# B&R Automation Studio project TD52 (part 18)

```c
/* Source: zlanhe.f */
#define zlanhe FORTRAN_WRAPPER(zlanhe)
extern double zlanhe(
    char   *norm,
    char   *uplo,
    ptrdiff_t *n,
    double *a,
    ptrdiff_t *lda,
    double *work
);

/* Source: zlanhf.f */
#define zlanhf FORTRAN_WRAPPER(zlanhf)
extern double zlanhf(
    char   *norm,
    char   *transr,
    char   *uplo,
    ptrdiff_t *n,
    double *a,
    double *work
);

/* Source: zlanhp.f */
#define zlanhp FORTRAN_WRAPPER(zlanhp)
extern double zlanhp(
    char   *norm,
    char   *uplo,
    ptrdiff_t *n,
    double *ap,
    double *work
);

/* Source: zlanhs.f */
#define zlanhs FORTRAN_WRAPPER(zlanhs)
extern double zlanhs(
    char   *norm,
    ptrdiff_t *n,
    double *a,
    ptrdiff_t *lda,
    double *work
);

/* Source: zlanht.f */
#define zlanht FORTRAN_WRAPPER(zlanht)
extern double zlanht(
    char   *norm,
    ptrdiff_t *n,
    double *d,
    double *e
);

/* Source: zlansb.f */
#define zlansb FORTRAN_WRAPPER(zlansb)
extern double zlansb(
    char   *norm,
    char   *uplo,
    ptrdiff_t *n,
    ptrdiff_t *k,
    double *ab,
    ptrdiff_t *ldab,
    double *work
);

/* Source: zlansp.f */
#define zlansp FORTRAN_WRAPPER(zlansp)
extern double zlansp(
    char   *norm,
    char   *uplo,
    ptrdiff_t *n,
    double *ap,
    double *work
);

/* Source: zlansy.f */
#define zlansy FORTRAN_WRAPPER(zlansy)
extern double zlansy(
    char   *norm,
    char   *uplo,
    ptrdiff_t *n,
    double *a,
    ptrdiff_t *lda,
    double *work
);

/* Source: zlantb.f */
#define zlantb FORTRAN_WRAPPER(zlantb)
extern double zlantb(
    char   *norm,
    char   *uplo,
    char   *diag,
    ptrdiff_t *n,
    ptrdiff_t *k,
    double *ab,
    ptrdiff_t *ldab,
    double *work
);

/* Source: zlantp.f */
#define zlantp FORTRAN_WRAPPER(zlantp)
extern double zlantp(
    char   *norm,
    char   *uplo,
    char   *diag,
    ptrdiff_t *n,
    double *ap,
    double *work
);

/* Source: zlantr.f */
#define zlantr FORTRAN_WRAPPER(zlantr)
extern double zlantr(
    char   *norm,
    char   *uplo,
    char   *diag,
    ptrdiff_t *m,
    ptrdiff_t *n,
    double *a,
    ptrdiff_t *lda,
    double *work
);

/* Source: zlapll.f */
#define zlapll FORTRAN_WRAPPER(zlapll)
extern void zlapll(
    ptrdiff_t *n,
    double *x,
    ptrdiff_t *incx,
    double *y,
    ptrdiff_t *incy,
    double *ssmin
);

/* Source: zlapmt.f */
#define zlapmt FORTRAN_WRAPPER(zlapmt)
extern void zlapmt(
    ptrdiff_t *forwrd,
    ptrdiff_t *m,
    ptrdiff_t *n,
    double *x,
    ptrdiff_t *ldx,
    ptrdiff_t *k
);

/* Source: zlaqgb.f */
#define zlaqgb FORTRAN_WRAPPER(zlaqgb)
extern void zlaqgb(
    ptrdiff_t *m,
    ptrdiff_t *n,
    ptrdiff_t *kl,
    ptrdiff_t *ku,
    double *ab,
    ptrdiff_t *ldab,
    double *r,
    double *c,
    double *rowcnd,
    double *colcnd,
    double *amax,
    char   *equed
);

/* Source: zlaqge.f */
#define zlaqge FORTRAN_WRAPPER(zlaqge)
extern void zlaqge(
    ptrdiff_t *m,
    ptrdiff_t *n,
    double *a,
    ptrdiff_t *lda,
    double *r,
    double *c,
    double *rowcnd,
    double *colcnd,
    double *amax,
    char   *equed
);

/* Source: zlaqhb.f */
#define zlaqhb FORTRAN_WRAPPER(zlaqhb)
extern void zlaqhb(
    char   *uplo,
    ptrdiff_t *n,
    ptrdiff_t *kd,
    double *ab,
    ptrdiff_t *ldab,
    double *s,
    double *scond,
    double *amax,
    char   *equed
);

/* Source: zlaqhe.f */
#define zlaqhe FORTRAN_WRAPPER(zlaqhe)
extern void zlaqhe(
    char   *uplo,
    ptrdiff_t *n,
    double *a,
    ptrdiff_t *lda,
    double *s,
    double *scond,
    double *amax,
    char   *equed
);

/* Source: zlaqhp.f */
#define zlaqhp FORTRAN_WRAPPER(zlaqhp)
extern void zlaqhp(
    char   *uplo,
    ptrdiff_t *n,
    double *ap,
    double *s,
    double *scond,
    double *amax,
    char   *equed
);

/* Source: zlaqp2.f */
#define zlaqp2 FORTRAN_WRAPPER(zlaqp2)
extern void zlaqp2(
    ptrdiff_t *m,
    ptrdiff_t *n,
    ptrdiff_t *offset,
    double *a,
    ptrdiff_t *lda,
    ptrdiff_t *jpvt,
    double *tau,
    double *vn1,
    double *vn2,
    double *work
);

/* Source: zlaqps.f */
#define zlaqps FORTRAN_WRAPPER(zlaqps)
extern void zlaqps(
    ptrdiff_t *m,
    ptrdiff_t *n,
    ptrdiff_t *offset,
    ptrdiff_t *nb,
    ptrdiff_t *kb,
    double *a,
    ptrdiff_t *lda,
    ptrdiff_t *jpvt,
    double *tau,
    double *vn1,
    double *vn2,
    double *auxv,
    double *f,
    ptrdiff_t *ldf
);

/* Source: zlaqr0.f */
#define zlaqr0 FORTRAN_WRAPPER(zlaqr0)
extern void zlaqr0(
    ptrdiff_t *wantt,
    ptrdiff_t *wantz,
    ptrdiff_t *n,
    ptrdiff_t *ilo,
    ptrdiff_t *ihi,
    double *h,
    ptrdiff_t *ldh,
    double *w,
    ptrdiff_t *iloz,
    ptrdiff_t *ihiz,
    double *z,
    ptrdiff_t *ldz,
    double *work,
    ptrdiff_t *lwork,
    ptrdiff_t *info
);

/* Source: zlaqr1.f */
#define zlaqr1 FORTRAN_WRAPPER(zlaqr1)
extern void zlaqr1(
    ptrdiff_t *n,
    double *h,
    ptrdiff_t *ldh,
    double *s1,
    double *s2,
    double *v
);

/* Source: zlaqr2.f */
#define zlaqr2 FORTRAN_WRAPPER(zlaqr2)
extern void zlaqr2(
    ptrdiff_t *wantt,
    ptrdiff_t *wantz,
    ptrdiff_t *n,
    ptrdiff_t *ktop,
    ptrdiff_t *kbot,
    ptrdiff_t *nw,
    double *h,
    ptrdiff_t *ldh,
    ptrdiff_t *iloz,
    ptrdiff_t *ihiz,
    double *z,
    ptrdiff_t *ldz,
    ptrdiff_t *ns,
    ptrdiff_t *nd,
    double *sh,
    double *v,
    ptrdiff_t *ldv,
    ptrdiff_t *nh,
    double *t,
    ptrdiff_t *ldt,
    ptrdiff_t *nv,
    double *wv,
    ptrdiff_t *ldwv,
    double *work,
    ptrdiff_t *lwork
);

/* Source: zlaqr3.f */
#define zlaqr3 FORTRAN_WRAPPER(zlaqr3)
extern void zlaqr3(
    ptrdiff_t *wantt,
    ptrdiff_t *wantz,
    ptrdiff_t *n,
    ptrdiff_t *ktop,
    ptrdiff_t *kbot,
    ptrdiff_t *nw,
    double *h,
    ptrdiff_t *ldh,
    ptrdiff_t *iloz,
    ptrdiff_t *ihiz,
    double *z,
    ptrdiff_t *ldz,
    ptrdiff_t *ns,
    ptrdiff_t *nd,
    double *sh,
    double *v,
    ptrdiff_t *ldv,
    ptrdiff_t *nh,
    double *t,
    ptrdiff_t *ldt,
    ptrdiff_t *nv,
    double *wv,
    ptrdiff_t *ldwv,
    double *work,
    ptrdiff_t *lwork
);

/* Source: zlaqr4.f */
#define zlaqr4 FORTRAN_WRAPPER(zlaqr4)
extern void zlaqr4(
    ptrdiff_t *wantt,
    ptrdiff_t *wantz,
    ptrdiff_t *n,
    ptrdiff_t *ilo,
    ptrdiff_t *ihi,
    double *h,
    ptrdiff_t *ldh,
    double *w,
    ptrdiff_t *iloz,
    ptrdiff_t *ihiz,
    double *z,
    ptrdiff_t *ldz,
    double *work,
    ptrdiff_t *lwork,
    ptrdiff_t *info
);

/* Source: zlaqr5.f */
#define zlaqr5 FORTRAN_WRAPPER(zlaqr5)
extern void zlaqr5(
    ptrdiff_t *wantt,
    ptrdiff_t *wantz,
    ptrdiff_t *kacc22,
    ptrdiff_t *n,
    ptrdiff_t *ktop,
    ptrdiff_t *kbot,
    ptrdiff_t *nshfts,
    double *s,
    double *h,
    ptrdiff_t *ldh,
    ptrdiff_t *iloz,
    ptrdiff_t *ihiz,
    double *z,
    ptrdiff_t *ldz,
    double *v,
    ptrdiff_t *ldv,
    double *u,
    ptrdiff_t *ldu,
    ptrdiff_t *nv,
    double *wv,
    ptrdiff_t *ldwv,
    ptrdiff_t *nh,
    double *wh,
    ptrdiff_t *ldwh
);

/* Source: zlaqsb.f */
#define zlaqsb FORTRAN_WRAPPER(zlaqsb)
extern void zlaqsb(
    char   *uplo,
    ptrdiff_t *n,
    ptrdiff_t *kd,
    double *ab,
    ptrdiff_t *ldab,
    double *s,
    double *scond,
    double *amax,
    char   *equed
);

/* Source: zlaqsp.f */
#define zlaqsp FORTRAN_WRAPPER(zlaqsp)
extern void zlaqsp(
    char   *uplo,
    ptrdiff_t *n,
    double *ap,
    double *s,
    double *scond,
    double *amax,
    char   *equed
);

/* Source: zlaqsy.f */
#define zlaqsy FORTRAN_WRAPPER(zlaqsy)
extern void zlaqsy(
    char   *uplo,
    ptrdiff_t *n,
    double *a,
    ptrdiff_t *lda,
    double *s,
    double *scond,
    double *amax,
    char   *equed
);

/* Source: zlar1v.f */
#define zlar1v FORTRAN_WRAPPER(zlar1v)
extern void zlar1v(
    ptrdiff_t *n,
    ptrdiff_t *b1,
    ptrdiff_t *bn,
    double *lambda,
    double *d,
    double *l,
    double *ld,
    double *lld,
    double *pivmin,
    double *gaptol,
    double *z,
    ptrdiff_t *wantnc,
    ptrdiff_t *negcnt,
    double *ztz,
    double *mingma,
    ptrdiff_t *r,
    ptrdiff_t *isuppz,
    double *nrminv,
    double *resid,
    double *rqcorr,
    double *work
);

/* Source: zlar2v.f */
#define zlar2v FORTRAN_WRAPPER(zlar2v)
extern void zlar2v(
    ptrdiff_t *n,
    double *x,
    double *y,
    double *z,
    ptrdiff_t *incx,
    double *c,
    double *s,
    ptrdiff_t *incc
);

/* Source: zlarcm.f */
#define zlarcm FORTRAN_WRAPPER(zlarcm)
extern void zlarcm(
    ptrdiff_t *m,
    ptrdiff_t *n,
    double *a,
    ptrdiff_t *lda,
    double *b,
    ptrdiff_t *ldb,
    double *c,
    ptrdiff_t *ldc,
    double *rwork
);

/* Source: zlarf.f */
#define zlarf FORTRAN_WRAPPER(zlarf)
extern void zlarf(
    char   *side,
    ptrdiff_t *m,
    ptrdiff_t *n,
    double *v,
    ptrdiff_t *incv,
    double *tau,
    double *c,
    ptrdiff_t *ldc,
    double *work
);

/* Source: zlarfb.f */
#define zlarfb FORTRAN_WRAPPER(zlarfb)
extern void zlarfb(
    char   *side,
    char   *trans,
    char   *direct,
    char   *storev,
    ptrdiff_t *m,
    ptrdiff_t *n,
    ptrdiff_t *k,
    double *v,
    ptrdiff_t *ldv,
    double *t,
    ptrdiff_t *ldt,
    double *c,
    ptrdiff_t *ldc,
    double *work,
    ptrdiff_t *ldwork
);

/* Source: zlarfg.f */
#define zlarfg FORTRAN_WRAPPER(zlarfg)
extern void zlarfg(
    ptrdiff_t *n,
    double *alpha,
    double *x,
    ptrdiff_t *incx,
    double *tau
);

/* Source: zlarfgp.f */
#define zlarfgp FORTRAN_WRAPPER(zlarfgp)
extern void zlarfgp(
    ptrdiff_t *n,
    double *alpha,
    double *x,
    ptrdiff_t *incx,
    double *tau
);

/* Source: zlarft.f */
#define zlarft FORTRAN_WRAPPER(zlarft)
extern void zlarft(
    char   *direct,
    char   *storev,
    ptrdiff_t *n,
    ptrdiff_t *k,
    double *v,
    ptrdiff_t *ldv,
    double *tau,
    double *t,
    ptrdiff_t *ldt
);

/* Source: zlarfx.f */
#define zlarfx FORTRAN_WRAPPER(zlarfx)
extern void zlarfx(
    char   *side,
    ptrdiff_t *m,
    ptrdiff_t *n,
    double *v,
    double *tau,
    double *c,
    ptrdiff_t *ldc,
    double *work
);

/* Source: zlargv.f */
#define zlargv FORTRAN_WRAPPER(zlargv)
extern void zlargv(
    ptrdiff_t *n,
    double *x,
    ptrdiff_t *incx,
    double *y,
    ptrdiff_t *incy,
    double *c,
    ptrdiff_t *incc
);

/* Source: zlarnv.f */
#define zlarnv FORTRAN_WRAPPER(zlarnv)
extern void zlarnv(
    ptrdiff_t *idist,
    ptrdiff_t *iseed,
    ptrdiff_t *n,
    double *x
);

/* Source: zlarrv.f */
#define zlarrv FORTRAN_WRAPPER(zlarrv)
extern void zlarrv(
    ptrdiff_t *n,
    double *vl,
    double *vu,
    double *d,
    double *l,
    double *pivmin,
    ptrdiff_t *isplit,
    ptrdiff_t *m,
    ptrdiff_t *dol,
    ptrdiff_t *dou,
    double *minrgp,
    double *rtol1,
    double *rtol2,
    double *w,
    double *werr,
    double *wgap,
    ptrdiff_t *iblock,
    ptrdiff_t *indexw,
    double *gers,
    double *z,
    ptrdiff_t *ldz,
    ptrdiff_t *isuppz,
    double *work,
    ptrdiff_t *iwork,
    ptrdiff_t *info
);

/* Source: zlartg.f */
#define zlartg FORTRAN_WRAPPER(zlartg)
extern void zlartg(
    double *f,
    double *g,
    double *cs,
    double *sn,
    double *r
);

/* Source: zlartv.f */
#define zlartv FORTRAN_WRAPPER(zlartv)
extern void zlartv(
    ptrdiff_t *n,
    double *x,
    ptrdiff_t *incx,
    double *y,
    ptrdiff_t *incy,
    double *c,
    double *s,
    ptrdiff_t *incc
);

/* Source: zlarz.f */
#define zlarz FORTRAN_WRAPPER(zlarz)
extern void zlarz(
    char   *side,
    ptrdiff_t *m,
    ptrdiff_t *n,
    ptrdiff_t *l,
    double *v,
    ptrdiff_t *incv,
    double *tau,
    double *c,
    ptrdiff_t *ldc,
    double *work
);

/* Source: zlarzb.f */
#define zlarzb FORTRAN_WRAPPER(zlarzb)
extern void zlarzb(
    char   *side,
    char   *trans,
    char   *direct,
    char   *storev,
    ptrdiff_t *m,
    ptrdiff_t *n,
    ptrdiff_t *k,
    ptrdiff_t *l,
    double *v,
    ptrdiff_t *ldv,
    double *t,
    ptrdiff_t *ldt,
    double *c,
    ptrdiff_t *ldc,
    double *work,
    ptrdiff_t *ldwork
);

/* Source: zlarzt.f */
#define zlarzt FORTRAN_WRAPPER(zlarzt)
extern void zlarzt(
    char   *direct,
    char   *storev,
    ptrdiff_t *n,
    ptrdiff_t *k,
    double *v,
    ptrdiff_t *ldv,
    double *tau,
    double *t,
    ptrdiff_t *ldt
);

/* Source: zlascl.f */
#define zlascl FORTRAN_WRAPPER(zlascl)
extern void zlascl(
    char   *type,
    ptrdiff_t *kl,
    ptrdiff_t *ku,
    double *cfrom,
    double *cto,
    ptrdiff_t *m,
    ptrdiff_t *n,
    double *a,
    ptrdiff_t *lda,
    ptrdiff_t *info
);

/* Source: zlaset.f */
#define zlaset FORTRAN_WRAPPER(zlaset)
extern void zlaset(
    char   *uplo,
    ptrdiff_t *m,
    ptrdiff_t *n,
    double *alpha,
    double *beta,
    double *a,
    ptrdiff_t *lda
);

/* Source: zlasr.f */
#define zlasr FORTRAN_WRAPPER(zlasr)
extern void zlasr(
    char   *side,
    char   *pivot,
    char   *direct,
    ptrdiff_t *m,
    ptrdiff_t *n,
    double *c,
    double *s,
    double *a,
    ptrdiff_t *lda
);

/* Source: zlassq.f */
#define zlassq FORTRAN_WRAPPER(zlassq)
extern void zlassq(
    ptrdiff_t *n,
    double *x,
    ptrdiff_t *incx,
    double *scale,
    double *sumsq
);

/* Source: zlaswp.f */
#define zlaswp FORTRAN_WRAPPER(zlaswp)
extern void zlaswp(
    ptrdiff_t *n,
    double *a,
    ptrdiff_t *lda,
    ptrdiff_t *k1,
    ptrdiff_t *k2,
    ptrdiff_t *ipiv,
    ptrdiff_t *incx
);

/* Source: zlasyf.f */
#define zlasyf FORTRAN_WRAPPER(zlasyf)
extern void zlasyf(
    char   *uplo,
    ptrdiff_t *n,
    ptrdiff_t *nb,
    ptrdiff_t *kb,
    double *a,
    ptrdiff_t *lda,
    ptrdiff_t *ipiv,
    double *w,
    ptrdiff_t *ldw,
    ptrdiff_t *info
);

/* Source: zlat2c.f */
#define zlat2c FORTRAN_WRAPPER(zlat2c)
extern void zlat2c(
    char   *uplo,
    ptrdiff_t *n,
    double *a,
    ptrdiff_t *lda,
    float  *sa,
    ptrdiff_t *ldsa,
    ptrdiff_t *info
);

/* Source: zlatbs.f */
#define zlatbs FORTRAN_WRAPPER(zlatbs)
extern void zlatbs(
    char   *uplo,
    char   *trans,
    char   *diag,
    char   *normin,
    ptrdiff_t *n,
    ptrdiff_t *kd,
    double *ab,
    ptrdiff_t *ldab,
    double *x,
    double *scale,
    double *cnorm,
    ptrdiff_t *info
);

/* Source: zlatdf.f */
#define zlatdf FORTRAN_WRAPPER(zlatdf)
extern void zlatdf(
    ptrdiff_t *ijob,
    ptrdiff_t *n,
    double *z,
    ptrdiff_t *ldz,
    double *rhs,
    double *rdsum,
    double *rdscal,
    ptrdiff_t *ipiv,
    ptrdiff_t *jpiv
);

/* Source: zlatps.f */
#define zlatps FORTRAN_WRAPPER(zlatps)
extern void zlatps(
    char   *uplo,
    char   *trans,
    char   *diag,
    char   *normin,
    ptrdiff_t *n,
    double *ap,
    double *x,
    double *scale,
    double *cnorm,
    ptrdiff_t *info
);

/* Source: zlatrd.f */
#define zlatrd FORTRAN_WRAPPER(zlatrd)
extern void zlatrd(
    char   *uplo,
    ptrdiff_t *n,
    ptrdiff_t *nb,
    double *a,
    ptrdiff_t *lda,
    double *e,
    double *tau,
    double *w,
    ptrdiff_t *ldw
);

/* Source: zlatrs.f */
#define zlatrs FORTRAN_WRAPPER(zlatrs)
extern void zlatrs(
    char   *uplo,
    char   *trans,
    char   *diag,
    char   *normin,
    ptrdiff_t *n,
    double *a,
    ptrdiff_t *lda,
    double *x,
    double *scale,
    double *cnorm,
    ptrdiff_t *info
);

/* Source: zlatrz.f */
#define zlatrz FORTRAN_WRAPPER(zlatrz)
extern void zlatrz(
    ptrdiff_t *m,
    ptrdiff_t *n,
    ptrdiff_t *l,
    double *a,
    ptrdiff_t *lda,
    double *tau,
    double *work
);

/* Source: zlatzm.f */
#define zlatzm FORTRAN_WRAPPER(zlatzm)
extern void zlatzm(
    char   *side,
    ptrdiff_t *m,
    ptrdiff_t *n,
    double *v,
    ptrdiff_t *incv,
    double *tau,
    double *c1,
    double *c2,
    ptrdiff_t *ldc,
    double *work
);

/* Source: zlauu2.f */
#define zlauu2 FORTRAN_WRAPPER(zlauu2)
extern void zlauu2(
    char   *uplo,
    ptrdiff_t *n,
    double *a,
    ptrdiff_t *lda,
    ptrdiff_t *info
);

/* Source: zlauum.f */
#define zlauum FORTRAN_WRAPPER(zlauum)
extern void zlauum(
    char   *uplo,
    ptrdiff_t *n,
    double *a,
    ptrdiff_t *lda,
    ptrdiff_t *info
);

/* Source: zpbcon.f */
#define zpbcon FORTRAN_WRAPPER(zpbcon)
extern void zpbcon(
    char   *uplo,
    ptrdiff_t *n,
    ptrdiff_t *kd,
    double *ab,
    ptrdiff_t *ldab,
    double *anorm,
    double *rcond,
    double *work,
    double *rwork,
    ptrdiff_t *info
);

/* Source: zpbequ.f */
#define zpbequ FORTRAN_WRAPPER(zpbequ)
extern void zpbequ(
    char   *uplo,
    ptrdiff_t *n,
    ptrdiff_t *kd,
    double *ab,
    ptrdiff_t *ldab,
    double *s,
    double *scond,
    double *amax,
    ptrdiff_t *info
);

/* Source: zpbrfs.f */
#define zpbrfs FORTRAN_WRAPPER(zpbrfs)
extern void zpbrfs(
    char   *uplo,
    ptrdiff_t *n,
    ptrdiff_t *kd,
    ptrdiff_t *nrhs,
    double *ab,
    ptrdiff_t *ldab,
    double *afb,
    ptrdiff_t *ldafb,
    double *b,
    ptrdiff_t *ldb,
    double *x,
    ptrdiff_t *ldx,
    double *ferr,
    double *berr,
    double *work,
    double *rwork,
    ptrdiff_t *info
);

/* Source: zpbstf.f */
#define zpbstf FORTRAN_WRAPPER(zpbstf)
extern void zpbstf(
    char   *uplo,
    ptrdiff_t *n,
    ptrdiff_t *kd,
    double *ab,
    ptrdiff_t *ldab,
    ptrdiff_t *info
);

/* Source: zpbsv.f */
#define zpbsv FORTRAN_WRAPPER(zpbsv)
extern void zpbsv(
    char   *uplo,
    ptrdiff_t *n,
    ptrdiff_t *kd,
    ptrdiff_t *nrhs,
    double *ab,
    ptrdiff_t *ldab,
    double *b,
    ptrdiff_t *ldb,
    ptrdiff_t *info
);

/* Source: zpbsvx.f */
#define zpbsvx FORTRAN_WRAPPER(zpbsvx)
extern void zpbsvx(
    char   *fact,
    char   *uplo,
    ptrdiff_t *n,
    ptrdiff_t *kd,
    ptrdiff_t *nrhs,
    double *ab,
    ptrdiff_t *ldab,
    double *afb,
    ptrdiff_t *ldafb,
    char   *equed,
    double *s,
    double *b,
    ptrdiff_t *ldb,
    double *x,
    ptrdiff_t *ldx,
    double *rcond,
    double *ferr,
    double *berr,
    double *work,
    double *rwork,
    ptrdiff_t *info
);

/* Source: zpbtf2.f */
#define zpbtf2 FORTRAN_WRAPPER(zpbtf2)
extern void zpbtf2(
    char   *uplo,
    ptrdiff_t *n,
    ptrdiff_t *kd,
    double *ab,
    ptrdiff_t *ldab,
    ptrdiff_t *info
);

/* Source: zpbtrf.f */
#define zpbtrf FORTRAN_WRAPPER(zpbtrf)
extern void zpbtrf(
    char   *uplo,
    ptrdiff_t *n,
    ptrdiff_t *kd,
    double *ab,
    ptrdiff_t *ldab,
    ptrdiff_t *info
);

/* Source: zpbtrs.f */
#define zpbtrs FORTRAN_WRAPPER(zpbtrs)
extern void zpbtrs(
    char   *uplo,
    ptrdiff_t *n,
    ptrdiff_t *kd,
    ptrdiff_t *nrhs,
    double *ab,
    ptrdiff_t *ldab,
    double *b,
    ptrdiff_t *ldb,
    ptrdiff_t *info
);

/* Source: zpftrf.f */
#define zpftrf FORTRAN_WRAPPER(zpftrf)
extern void zpftrf(
    char   *transr,
    char   *uplo,
    ptrdiff_t *n,
    double *a,
    ptrdiff_t *info
);

/* Source: zpftri.f */
#define zpftri FORTRAN_WRAPPER(zpftri)
extern void zpftri(
    char   *transr,
    char   *uplo,
    ptrdiff_t *n,
    double *a,
    ptrdiff_t *info
);

/* Source: zpftrs.f */
#define zpftrs FORTRAN_WRAPPER(zpftrs)
extern void zpftrs(
    char   *transr,
    char   *uplo,
    ptrdiff_t *n,
    ptrdiff_t *nrhs,
    double *a,
    double *b,
    ptrdiff_t *ldb,
    ptrdiff_t *info
);

/* Source: zpocon.f */
#define zpocon FORTRAN_WRAPPER(zpocon)
extern void zpocon(
    char   *uplo,
    ptrdiff_t *n,
    double *a,
    ptrdiff_t *lda,
    double *anorm,
    double *rcond,
    double *work,
    double *rwork,
    ptrdiff_t *info
);

/* Source: zpoequ.f */
#define zpoequ FORTRAN_WRAPPER(zpoequ)
extern void zpoequ(
    ptrdiff_t *n,
    double *a,
    ptrdiff_t *lda,
    double *s,
    double *scond,
    double *amax,
    ptrdiff_t *info
);

/* Source: zpoequb.f */
#define zpoequb FORTRAN_WRAPPER(zpoequb)
extern void zpoequb(
    ptrdiff_t *n,
    double *a,
    ptrdiff_t *lda,
    double *s,
    double *scond,
    double *amax,
    ptrdiff_t *info
);

/* Source: zporfs.f */
#define zporfs FORTRAN_WRAPPER(zporfs)
extern void zporfs(
    char   *uplo,
    ptrdiff_t *n,
    ptrdiff_t *nrhs,
    double *a,
    ptrdiff_t *lda,
    double *af,
    ptrdiff_t *ldaf,
    double *b,
    ptrdiff_t *ldb,
    double *x,
    ptrdiff_t *ldx,
    double *ferr,
    double *berr,
    double *work,
    double *rwork,
    ptrdiff_t *info
);

/* Source: zposv.f */
#define zposv FORTRAN_WRAPPER(zposv)
extern void zposv(
    char   *uplo,
    ptrdiff_t *n,
    ptrdiff_t *nrhs,
    double *a,
    ptrdiff_t *lda,
    double *b,
    ptrdiff_t *ldb,
    ptrdiff_t *info
);

/* Source: zposvx.f */
#define zposvx FORTRAN_WRAPPER(zposvx)
extern void zposvx(
    char   *fact,
    char   *uplo,
    ptrdiff_t *n,
    ptrdiff_t *nrhs,
    double *a,
    ptrdiff_t *lda,
    double *af,
    ptrdiff_t *ldaf,
    char   *equed,
    double *s,
    double *b,
    ptrdiff_t *ldb,
    double *x,
    ptrdiff_t *ldx,
    double *rcond,
    double *ferr,
    double *berr,
    double *work,
    double *rwork,
    ptrdiff_t *info
);

/* Source: zpotf2.f */
#define zpotf2 FORTRAN_WRAPPER(zpotf2)
extern void zpotf2(
    char   *uplo,
    ptrdiff_t *n,
    double *a,
    ptrdiff_t *lda,
    ptrdiff_t *info
);

/* Source: zpotrf.f */
#define zpotrf FORTRAN_WRAPPER(zpotrf)
extern void zpotrf(
    char   *uplo,
    ptrdiff_t *n,
    double *a,
    ptrdiff_t *lda,
    ptrdiff_t *info
);

/* Source: zpotri.f */
#define zpotri FORTRAN_WRAPPER(zpotri)
extern void zpotri(
    char   *uplo,
    ptrdiff_t *n,
    double *a,
    ptrdiff_t *lda,
    ptrdiff_t *info
);

/* Source: zpotrs.f */
#define zpotrs FORTRAN_WRAPPER(zpotrs)
extern void zpotrs(
    char   *uplo,
    ptrdiff_t *n,
    ptrdiff_t *nrhs,
    double *a,
    ptrdiff_t *lda,
    double *b,
    ptrdiff_t *ldb,
    ptrdiff_t *info
);

/* Source: zppcon.f */
#define zppcon FORTRAN_WRAPPER(zppcon)
extern void zppcon(
    char   *uplo,
    ptrdiff_t *n,
    double *ap,
    double *anorm,
    double *rcond,
    double *work,
    double *rwork,
    ptrdiff_t *info
);

/* Source: zppequ.f */
#define zppequ FORTRAN_WRAPPER(zppequ)
extern void zppequ(
    char   *uplo,
    ptrdiff_t *n,
    double *ap,
    double *s,
    double *scond,
    double *amax,
    ptrdiff_t *info
);

/* Source: zpprfs.f */
#define zpprfs FORTRAN_WRAPPER(zpprfs)
extern void zpprfs(
    char   *uplo,
    ptrdiff_t *n,
    ptrdiff_t *nrhs,
    double *ap,
    double *afp,
    double *b,
    ptrdiff_t *ldb,
    double *x,
    ptrdiff_t *ldx,
    double *ferr,
    double *berr,
    double *work,
    double *rwork,
    ptrdiff_t *info
);

/* Source: zppsv.f */
#define zppsv FORTRAN_WRAPPER(zppsv)
extern void zppsv(
    char   *uplo,
    ptrdiff_t *n,
    ptrdiff_t *nrhs,
    double *ap,
    double *b,
    ptrdiff_t *ldb,
    ptrdiff_t *info
);

/* Source: zppsvx.f */
#define zppsvx FORTRAN_WRAPPER(zppsvx)
extern void zppsvx(
    char   *fact,
    char   *uplo,
    ptrdiff_t *n,
    ptrdiff_t *nrhs,
    double *ap,
    double *afp,
    char   *equed,
    double *s,
    double *b,
    ptrdiff_t *ldb,
    double *x,
    ptrdiff_t *ldx,
    double *rcond,
    double *ferr,
    double *berr,
    double *work,
    double *rwork,
    ptrdiff_t *info
);

/* Source: zpptrf.f */
#define zpptrf FORTRAN_WRAPPER(zpptrf)
extern void zpptrf(
    char   *uplo,
    ptrdiff_t *n,
    double *ap,
    ptrdiff_t *info
);

/* Source: zpptri.f */
#define zpptri FORTRAN_WRAPPER(zpptri)
extern void zpptri(
    char   *uplo,
    ptrdiff_t *n,
    double *ap,
    ptrdiff_t *info
);

/* Source: zpptrs.f */
#define zpptrs FORTRAN_WRAPPER(zpptrs)
extern void zpptrs(
    char   *uplo,
    ptrdiff_t *n,
    ptrdiff_t *nrhs,
    double *ap,
    double *b,
    ptrdiff_t *ldb,
    ptrdiff_t *info
);

/* Source: zpstf2.f */
#define zpstf2 FORTRAN_WRAPPER(zpstf2)
extern void zpstf2(
    char   *uplo,
    ptrdiff_t *n,
    double *a,
    ptrdiff_t *lda,
    ptrdiff_t *piv,
    ptrdiff_t *rank,
    double *tol,
    double *work,
    ptrdiff_t *info
);

/* Source: zpstrf.f */
#define zpstrf FORTRAN_WRAPPER(zpstrf)
extern void zpstrf(
    char   *uplo,
    ptrdiff_t *n,
    double *a,
    ptrdiff_t *lda,
    ptrdiff_t *piv,
    ptrdiff_t *rank,
    double *tol,
    double *work,
    ptrdiff_t *info
);

/* Source: zptcon.f */
#define zptcon FORTRAN_WRAPPER(zptcon)
extern void zptcon(
    ptrdiff_t *n,
    double *d,
    double *e,
    double *anorm,
    double *rcond,
    double *rwork,
    ptrdiff_t *info
);

/* Source: zpteqr.f */
#define zpteqr FORTRAN_WRAPPER(zpteqr)
extern void zpteqr(
    char   *compz,
    ptrdiff_t *n,
    double *d,
    double *e,
    double *z,
    ptrdiff_t *ldz,
    double *work,
    ptrdiff_t *info
);

/* Source: zptrfs.f */
#define zptrfs FORTRAN_WRAPPER(zptrfs)
extern void zptrfs(
    char   *uplo,
    ptrdiff_t *n,
    ptrdiff_t *nrhs,
    double *d,
    double *e,
    double *df,
    double *ef,
    double *b,
    ptrdiff_t *ldb,
    double *x,
    ptrdiff_t *ldx,
    double *ferr,
    double *berr,
    double *work,
    double *rwork,
    ptrdiff_t *info
);

/* Source: zptsv.f */
#define zptsv FORTRAN_WRAPPER(zptsv)
extern void zptsv(
    ptrdiff_t *n,
    ptrdiff_t *nrhs,
    double *d,
    double *e,
    double *b,
    ptrdiff_t *ldb,
    ptrdiff_t *info
);

/* Source: zptsvx.f */
#define zptsvx FORTRAN_WRAPPER(zptsvx)
extern void zptsvx(
    char   *fact,
    ptrdiff_t *n,
    ptrdiff_t *nrhs,
    double *d,
    double *e,
    double *df,
    double *ef,
    double *b,
    ptrdiff_t *ldb,
    double *x,
    ptrdiff_t *ldx,
    double *rcond,
    double *ferr,
    double *berr,
    double *work,
    double *rwork,
    ptrdiff_t *info
);

/* Source: zpttrf.f */
#define zpttrf FORTRAN_WRAPPER(zpttrf)
extern void zpttrf(
    ptrdiff_t *n,
    double *d,
    double *e,
    ptrdiff_t *info
);

/* Source: zpttrs.f */
#define zpttrs FORTRAN_WRAPPER(zpttrs)
extern void zpttrs(
    char   *uplo,
    ptrdiff_t *n,
    ptrdiff_t *nrhs,
    double *d,
    double *e,
    double *b,
    ptrdiff_t *ldb,
    ptrdiff_t *info
);

/* Source: zptts2.f */
#define zptts2 FORTRAN_WRAPPER(zptts2)
extern void zptts2(
    ptrdiff_t *iuplo,
    ptrdiff_t *n,
    ptrdiff_t *nrhs,
    double *d,
    double *e,
    double *b,
    ptrdiff_t *ldb
);

/* Source: zrot.f */
#define zrot FORTRAN_WRAPPER(zrot)
extern void zrot(
    ptrdiff_t *n,
    double *cx,
    ptrdiff_t *incx,
    double *cy,
    ptrdiff_t *incy,
    double *c,
    double *s
);

/* Source: zspcon.f */
#define zspcon FORTRAN_WRAPPER(zspcon)
extern void zspcon(
    char   *uplo,
    ptrdiff_t *n,
    double *ap,
    ptrdiff_t *ipiv,
    double *anorm,
    double *rcond,
    double *work,
    ptrdiff_t *info
);

/* Source: zspmv.f */
#define zspmv FORTRAN_WRAPPER(zspmv)
extern void zspmv(
    char   *uplo,
    ptrdiff_t *n,
    double *alpha,
    double *ap,
    double *x,
    ptrdiff_t *incx,
    double *beta,
    double *y,
    ptrdiff_t *incy
);

/* Source: zspr.f */
#define zspr FORTRAN_WRAPPER(zspr)
extern void zspr(
    char   *uplo,
    ptrdiff_t *n,
    double *alpha,
    double *x,
    ptrdiff_t *incx,
    double *ap
);

/* Source: zsprfs.f */
#define zsprfs FORTRAN_WRAPPER(zsprfs)
extern void zsprfs(
    char   *uplo,
    ptrdiff_t *n,
    ptrdiff_t *nrhs,
    double *ap,
    double *afp,
    ptrdiff_t *ipiv,
    double *b,
    ptrdiff_t *ldb,
    double *x,
    ptrdiff_t *ldx,
    double *ferr,
    double *berr,
    double *work,
    double *rwork,
    ptrdiff_t *info
);

/* Source: zspsv.f */
#define zspsv FORTRAN_WRAPPER(zspsv)
extern void zspsv(
    char   *uplo,
    ptrdiff_t *n,
    ptrdiff_t *nrhs,
    double *ap,
    ptrdiff_t *ipiv,
    double *b,
    ptrdiff_t *ldb,
    ptrdiff_t *info
);

/* Source: zspsvx.f */
#define zspsvx FORTRAN_WRAPPER(zspsvx)
extern void zspsvx(
    char   *fact,
    char   *uplo,
    ptrdiff_t *n,
    ptrdiff_t *nrhs,
    double *ap,
    double *afp,
    ptrdiff_t *ipiv,
    double *b,
    ptrdiff_t *ldb,
    double *x,
    ptrdiff_t *ldx,
    double *rcond,
    double *ferr,
    double *berr,
    double *work,
    double *rwork,
    ptrdiff_t *info
);

/* Source: zsptrf.f */
#define zsptrf FORTRAN_WRAPPER(zsptrf)
extern void zsptrf(
    char   *uplo,
    ptrdiff_t *n,
    double *ap,
    ptrdiff_t *ipiv,
    ptrdiff_t *info
);

/* Source: zsptri.f */
#define zsptri FORTRAN_WRAPPER(zsptri)
extern void zsptri(
    char   *uplo,
    ptrdiff_t *n,
    double *ap,
    ptrdiff_t *ipiv,
    double *work,
    ptrdiff_t *info
);

/* Source: zsptrs.f */
#define zsptrs FORTRAN_WRAPPER(zsptrs)
extern void zsptrs(
    char   *uplo,
    ptrdiff_t *n,
    ptrdiff_t *nrhs,
    double *ap,
    ptrdiff_t *ipiv,
    double *b,
    ptrdiff_t *ldb,
    ptrdiff_t *info
);

/* Source: zstedc.f */
#define zstedc FORTRAN_WRAPPER(zstedc)
extern void zstedc(
    char   *compz,
    ptrdiff_t *n,
    double *d,
    double *e,
    double *z,
    ptrdiff_t *ldz,
    double *work,
    ptrdiff_t *lwork,
    double *rwork,
    ptrdiff_t *lrwork,
    ptrdiff_t *iwork,
    ptrdiff_t *liwork,
    ptrdiff_t *info
);

/* Source: zstegr.f */
#define zstegr FORTRAN_WRAPPER(zstegr)
extern void zstegr(
    char   *jobz,
    char   *range,
    ptrdiff_t *n,
    double *d,
    double *e,
    double *vl,
    double *vu,
    ptrdiff_t *il,
    ptrdiff_t *iu,
    double *abstol,
    ptrdiff_t *m,
    double *w,
    double *z,
    ptrdiff_t *ldz,
    ptrdiff_t *isuppz,
    double *work,
    ptrdiff_t *lwork,
    ptrdiff_t *iwork,
    ptrdiff_t *liwork,
    ptrdiff_t *info
);

/* Source: zstein.f */
#define zstein FORTRAN_WRAPPER(zstein)
extern void zstein(
    ptrdiff_t *n,
    double *d,
    double *e,
    ptrdiff_t *m,
    double *w,
    ptrdiff_t *iblock,
    ptrdiff_t *isplit,
    double *z,
    ptrdiff_t *ldz,
    double *work,
    ptrdiff_t *iwork,
    ptrdiff_t *ifail,
    ptrdiff_t *info
);

/* Source: zstemr.f */
#define zstemr FORTRAN_WRAPPER(zstemr)
extern void zstemr(
    char   *jobz,
    char   *range,
    ptrdiff_t *n,
    double *d,
    double *e,
    double *vl,
    double *vu,
    ptrdiff_t *il,
    ptrdiff_t *iu,
    ptrdiff_t *m,
    double *w,
    double *z,
    ptrdiff_t *ldz,
    ptrdiff_t *nzc,
    ptrdiff_t *isuppz,
    ptrdiff_t *tryrac,
    double *work,
    ptrdiff_t *lwork,
    ptrdiff_t *iwork,
    ptrdiff_t *liwork,
    ptrdiff_t *info
);

/* Source: zsteqr.f */
#define zsteqr FORTRAN_WRAPPER(zsteqr)
extern void zsteqr(
    char   *compz,
    ptrdiff_t *n,
    double *d,
    double *e,
    double *z,
    ptrdiff_t *ldz,
    double *work,
    ptrdiff_t *info
);

/* Source: zsycon.f */
#define zsycon FORTRAN_WRAPPER(zsycon)
extern void zsycon(
    char   *uplo,
    ptrdiff_t *n,
    double *a,
    ptrdiff_t *lda,
    ptrdiff_t *ipiv,
    double *anorm,
    double *rcond,
    double *work,
    ptrdiff_t *info
);

/* Source: zsyequb.f */
#define zsyequb FORTRAN_WRAPPER(zsyequb)
extern void zsyequb(
    char   *uplo,
    ptrdiff_t *n,
    double *a,
    ptrdiff_t *lda,
    double *s,
    double *scond,
    double *amax,
    double *work,
    ptrdiff_t *info
);

/* Source: zsymv.f */
#define zsymv FORTRAN_WRAPPER(zsymv)
extern void zsymv(
    char   *uplo,
    ptrdiff_t *n,
    double *alpha,
    double *a,
    ptrdiff_t *lda,
    double *x,
    ptrdiff_t *incx,
    double *beta,
    double *y,
    ptrdiff_t *incy
);

/* Source: zsyr.f */
#define zsyr FORTRAN_WRAPPER(zsyr)
extern void zsyr(
    char   *uplo,
    ptrdiff_t *n,
    double *alpha,
    double *x,
    ptrdiff_t *incx,
    double *a,
    ptrdiff_t *lda
);

/* Source: zsyrfs.f */
#define zsyrfs FORTRAN_WRAPPER(zsyrfs)
extern void zsyrfs(
    char   *uplo,
    ptrdiff_t *n,
    ptrdiff_t *nrhs,
    double *a,
    ptrdiff_t *lda,
    double *af,
    ptrdiff_t *ldaf,
    ptrdiff_t *ipiv,
    double *b,
    ptrdiff_t *ldb,
    double *x,
    ptrdiff_t *ldx,
    double *ferr,
    double *berr,
    double *work,
    double *rwork,
    ptrdiff_t *info
);

/* Source: zsysv.f */
#define zsysv FORTRAN_WRAPPER(zsysv)
extern void zsysv(
    char   *uplo,
    ptrdiff_t *n,
    ptrdiff_t *nrhs,
    double *a,
    ptrdiff_t *lda,
    ptrdiff_t *ipiv,
    double *b,
    ptrdiff_t *ldb,
    double *work,
    ptrdiff_t *lwork,
    ptrdiff_t *info
);

/* Source: zsysvx.f */
#define zsysvx FORTRAN_WRAPPER(zsysvx)
extern void zsysvx(
    char   *fact,
    char   *uplo,
    ptrdiff_t *n,
    ptrdiff_t *nrhs,
    double *a,
    ptrdiff_t *lda,
    double *af,
    ptrdiff_t *ldaf,
    ptrdiff_t *ipiv,
    double *b,
    ptrdiff_t *ldb,
    double *x,
    ptrdiff_t *ldx,
    double *rcond,
    double *ferr,
    double *berr,
    double *work,
    ptrdiff_t *lwork,
    double *rwork,
    ptrdiff_t *info
);

/* Source: zsytf2.f */
#define zsytf2 FORTRAN_WRAPPER(zsytf2)
extern void zsytf2(
    char   *uplo,
    ptrdiff_t *n,
    double *a,
    ptrdiff_t *lda,
    ptrdiff_t *ipiv,
    ptrdiff_t *info
);

/* Source: zsytrf.f */
#define zsytrf FORTRAN_WRAPPER(zsytrf)
extern void zsytrf(
    char   *uplo,
    ptrdiff_t *n,
    double *a,
    ptrdiff_t *lda,
    ptrdiff_t *ipiv,
    double *work,
    ptrdiff_t *lwork,
    ptrdiff_t *info
);

/* Source: zsytri.f */
#define zsytri FORTRAN_WRAPPER(zsytri)
extern void zsytri(
    char   *uplo,
    ptrdiff_t *n,
    double *a,
    ptrdiff_t *lda,
    ptrdiff_t *ipiv,
    double *work,
    ptrdiff_t *info
);

/* Source: zsytrs.f */
#define zsytrs FORTRAN_WRAPPER(zsytrs)
extern void zsytrs(
    char   *uplo,
    ptrdiff_t *n,
    ptrdiff_t *nrhs,
    double *a,
    ptrdiff_t *lda,
    ptrdiff_t *ipiv,
    double *b,
    ptrdiff_t *ldb,
    ptrdiff_t *info
);

/* Source: ztbcon.f */
#define ztbcon FORTRAN_WRAPPER(ztbcon)
extern void ztbcon(
    char   *norm,
    char   *uplo,
    char   *diag,
    ptrdiff_t *n,
    ptrdiff_t *kd,
    double *ab,
    ptrdiff_t *ldab,
    double *rcond,
    double *work,
    double *rwork,
    ptrdiff_t *info
);

/* Source: ztbrfs.f */
#define ztbrfs FORTRAN_WRAPPER(ztbrfs)
extern void ztbrfs(
    char   *uplo,
    char   *trans,
    char   *diag,
    ptrdiff_t *n,
    ptrdiff_t *kd,
    ptrdiff_t *nrhs,
    double *ab,
    ptrdiff_t *ldab,
    double *b,
    ptrdiff_t *ldb,
    double *x,
    ptrdiff_t *ldx,
    double *ferr,
    double *berr,
    double *work,
    double *rwork,
    ptrdiff_t *info
);

/* Source: ztbtrs.f */
#define ztbtrs FORTRAN_WRAPPER(ztbtrs)
extern void ztbtrs(
    char   *uplo,
    char   *trans,
    char   *diag,
    ptrdiff_t *n,
    ptrdiff_t *kd,
    ptrdiff_t *nrhs,
    double *ab,
    ptrdiff_t *ldab,
    double *b,
    ptrdiff_t *ldb,
    ptrdiff_t *info
);

/* Source: ztfsm.f */
#define ztfsm FORTRAN_WRAPPER(ztfsm)
extern void ztfsm(
    char   *transr,
    char   *side,
    char   *uplo,
    char   *trans,
    char   *diag,
    ptrdiff_t *m,
    ptrdiff_t *n,
    double *alpha,
    double *a,
    double *b,
    ptrdiff_t *ldb
);

/* Source: ztftri.f */
#define ztftri FORTRAN_WRAPPER(ztftri)
extern void ztftri(
    char   *transr,
    char   *uplo,
    char   *diag,
    ptrdiff_t *n,
    double *a,
    ptrdiff_t *info
);

/* Source: ztfttp.f */
#define ztfttp FORTRAN_WRAPPER(ztfttp)
extern void ztfttp(
    char   *transr,
    char   *uplo,
    ptrdiff_t *n,
    double *arf,
    double *ap,
    ptrdiff_t *info
);

/* Source: ztfttr.f */
#define ztfttr FORTRAN_WRAPPER(ztfttr)
extern void ztfttr(
    char   *transr,
    char   *uplo,
    ptrdiff_t *n,
    double *arf,
    double *a,
    ptrdiff_t *lda,
    ptrdiff_t *info
);

/* Source: ztgevc.f */
#define ztgevc FORTRAN_WRAPPER(ztgevc)
extern void ztgevc(
    char   *side,
    char   *howmny,
    ptrdiff_t *select,
    ptrdiff_t *n,
    double *s,
    ptrdiff_t *lds,
    double *p,
    ptrdiff_t *ldp,
    double *vl,
    ptrdiff_t *ldvl,
    double *vr,
    ptrdiff_t *ldvr,
    ptrdiff_t *mm,
    ptrdiff_t *m,
    double *work,
    double *rwork,
    ptrdiff_t *info
);

/* Source: ztgex2.f */
#define ztgex2 FORTRAN_WRAPPER(ztgex2)
extern void ztgex2(
    ptrdiff_t *wantq,
    ptrdiff_t *wantz,
    ptrdiff_t *n,
    double *a,
    ptrdiff_t *lda,
    double *b,
    ptrdiff_t *ldb,
    double *q,
    ptrdiff_t *ldq,
    double *z,
    ptrdiff_t *ldz,
    ptrdiff_t *j1_,
    ptrdiff_t *info
);

/* Source: ztgexc.f */
#define ztgexc FORTRAN_WRAPPER(ztgexc)
extern void ztgexc(
    ptrdiff_t *wantq,
    ptrdiff_t *wantz,
    ptrdiff_t *n,
    double *a,
    ptrdiff_t *lda,
    double *b,
    ptrdiff_t *ldb,
    double *q,
    ptrdiff_t *ldq,
    double *z,
    ptrdiff_t *ldz,
    ptrdiff_t *ifst,
    ptrdiff_t *ilst,
    ptrdiff_t *info
);

/* Source: ztgsen.f */
#define ztgsen FORTRAN_WRAPPER(ztgsen)
extern void ztgsen(
    ptrdiff_t *ijob,
    ptrdiff_t *wantq,
    ptrdiff_t *wantz,
    ptrdiff_t *select,
    ptrdiff_t *n,
    double *a,
    ptrdiff_t *lda,
    double *b,
    ptrdiff_t *ldb,
    double *alpha,
    double *beta,
    double *q,
    ptrdiff_t *ldq,
    double *z,
    ptrdiff_t *ldz,
    ptrdiff_t *m,
    double *pl,
    double *pr,
    double *dif,
    double *work,
    ptrdiff_t *lwork,
    ptrdiff_t *iwork,
    ptrdiff_t *liwork,
    ptrdiff_t *info
);

/* Source: ztgsja.f */
#define ztgsja FORTRAN_WRAPPER(ztgsja)
extern void ztgsja(
    char   *jobu,
    char   *jobv,
    char   *jobq,
    ptrdiff_t *m,
    ptrdiff_t *p,
    ptrdiff_t *n,
    ptrdiff_t *k,
    ptrdiff_t *l,
    double *a,
    ptrdiff_t *lda,
    double *b,
    ptrdiff_t *ldb,
    double *tola,
    double *tolb,
    double *alpha,
    double *beta,
    double *u,
    ptrdiff_t *ldu,
    double *v,
    ptrdiff_t *ldv,
    double *q,
    ptrdiff_t *ldq,
    double *work,
    ptrdiff_t *ncycle,
    ptrdiff_t *info
);

/* Source: ztgsna.f */
#define ztgsna FORTRAN_WRAPPER(ztgsna)
extern void ztgsna(
    char   *job,
    char   *howmny,
    ptrdiff_t *select,
    ptrdiff_t *n,
    double *a,
    ptrdiff_t *lda,
    double *b,
    ptrdiff_t *ldb,
    double *vl,
    ptrdiff_t *ldvl,
    double *vr,
    ptrdiff_t *ldvr,
    double *s,
    double *dif,
    ptrdiff_t *mm,
    ptrdiff_t *m,
    double *work,
    ptrdiff_t *lwork,
    ptrdiff_t *iwork,
    ptrdiff_t *info
);

/* Source: ztgsy2.f */
#define ztgsy2 FORTRAN_WRAPPER(ztgsy2)
extern void ztgsy2(
    char   *trans,
    ptrdiff_t *ijob,
    ptrdiff_t *m,
    ptrdiff_t *n,
    double *a,
    ptrdiff_t *lda,
    double *b,
    ptrdiff_t *ldb,
    double *c,
    ptrdiff_t *ldc,
    double *d,
    ptrdiff_t *ldd,
    double *e,
    ptrdiff_t *lde,
    double *f,
    ptrdiff_t *ldf,
    double *scale,
    double *rdsum,
    double *rdscal,
    ptrdiff_t *info
);

/* Source: ztgsyl.f */
#define ztgsyl FORTRAN_WRAPPER(ztgsyl)
extern void ztgsyl(
    char   *trans,
    ptrdiff_t *ijob,
    ptrdiff_t *m,
    ptrdiff_t *n,
    double *a,
    ptrdiff_t *lda,
    double *b,
    ptrdiff_t *ldb,
    double *c,
    ptrdiff_t *ldc,
    double *d,
    ptrdiff_t *ldd,
    double *e,
    ptrdiff_t *lde,
    double *f,
    ptrdiff_t *ldf,
    double *scale,
    double *dif,
    double *work,
    ptrdiff_t *lwork,
    ptrdiff_t *iwork,
    ptrdiff_t *info
);

/* Source: ztpcon.f */
#define ztpcon FORTRAN_WRAPPER(ztpcon)
extern void ztpcon(
    char   *norm,
    char   *uplo,
    char   *diag,
    ptrdiff_t *n,
    double *ap,
    double *rcond,
    double *work,
    double *rwork,
    ptrdiff_t *info
);

/* Source: ztprfs.f */
#define ztprfs FORTRAN_WRAPPER(ztprfs)
extern void ztprfs(
    char   *uplo,
    char   *trans,
    char   *diag,
    ptrdiff_t *n,
    ptrdiff_t *nrhs,
    double *ap,
    double *b,
    ptrdiff_t *ldb,
    double *x,
    ptrdiff_t *ldx,
    double *ferr,
    double *berr,
    double *work,
    double *rwork,
    ptrdiff_t *info
);

/* Source: ztptri.f */
#define ztptri FORTRAN_WRAPPER(ztptri)
extern void ztptri(
    char   *uplo,
    char   *diag,
    ptrdiff_t *n,
    double *ap,
    ptrdiff_t *info
);

/* Source: ztptrs.f */
#define ztptrs FORTRAN_WRAPPER(ztptrs)
extern void ztptrs(
    char   *uplo,
    char   *trans,
    char   *diag,
    ptrdiff_t *n,
    ptrdiff_t *nrhs,
    double *ap,
    double *b,
    ptrdiff_t *ldb,
    ptrdiff_t *info
);

/* Source: ztpttf.f */
#define ztpttf FORTRAN_WRAPPER(ztpttf)
extern void ztpttf(
    char   *transr,
    char   *uplo,
    ptrdiff_t *n,
    double *ap,
    double *arf,
    ptrdiff_t *info
);

/* Source: ztpttr.f */
#define ztpttr FORTRAN_WRAPPER(ztpttr)
extern void ztpttr(
    char   *uplo,
    ptrdiff_t *n,
    double *ap,
    double *a,
    ptrdiff_t *lda,
    ptrdiff_t *info
);

/* Source: ztrcon.f */
#define ztrcon FORTRAN_WRAPPER(ztrcon)
extern void ztrcon(
    char   *norm,
    char   *uplo,
    char   *diag,
    ptrdiff_t *n,
    double *a,
    ptrdiff_t *lda,
    double *rcond,
    double *work,
    double *rwork,
    ptrdiff_t *info
);

/* Source: ztrevc.f */
#define ztrevc FORTRAN_WRAPPER(ztrevc)
extern void ztrevc(
    char   *side,
    char   *howmny,
    ptrdiff_t *select,
    ptrdiff_t *n,
    double *t,
    ptrdiff_t *ldt,
    double *vl,
    ptrdiff_t *ldvl,
    double *vr,
    ptrdiff_t *ldvr,
    ptrdiff_t *mm,
    ptrdiff_t *m,
    double *work,
    double *rwork,
    ptrdiff_t *info
);

/* Source: ztrexc.f */
#define ztrexc FORTRAN_WRAPPER(ztrexc)
extern void ztrexc(
    char   *compq,
    ptrdiff_t *n,
    double *t,
    ptrdiff_t *ldt,
    double *q,
    ptrdiff_t *ldq,
    ptrdiff_t *ifst,
    ptrdiff_t *ilst,
    ptrdiff_t *info
);

/* Source: ztrrfs.f */
#define ztrrfs FORTRAN_WRAPPER(ztrrfs)
extern void ztrrfs(
    char   *uplo,
    char   *trans,
    char   *diag,
    ptrdiff_t *n,
    ptrdiff_t *nrhs,
    double *a,
    ptrdiff_t *lda,
    double *b,
    ptrdiff_t *ldb,
    double *x,
    ptrdiff_t *ldx,
    double *ferr,
    double *berr,
    double *work,
    double *rwork,
    ptrdiff_t *info
);

/* Source: ztrsen.f */
#define ztrsen FORTRAN_WRAPPER(ztrsen)
extern void ztrsen(
    char   *job,
    char   *compq,
    ptrdiff_t *select,
    ptrdiff_t *n,
    double *t,
    ptrdiff_t *ldt,
    double *q,
    ptrdiff_t *ldq,
    double *w,
    ptrdiff_t *m,
    double *s,
    double *sep,
    double *work,
    ptrdiff_t *lwork,
    ptrdiff_t *info
);

/* Source: ztrsna.f */
#define ztrsna FORTRAN_WRAPPER(ztrsna)
extern void ztrsna(
    char   *job,
    char   *howmny,
    ptrdiff_t *select,
    ptrdiff_t *n,
    double *t,
    ptrdiff_t *ldt,
    double *vl,
    ptrdiff_t *ldvl,
    double *vr,
    ptrdiff_t *ldvr,
    double *s,
    double *sep,
    ptrdiff_t *mm,
    ptrdiff_t *m,
    double *work,
    ptrdiff_t *ldwork,
    double *rwork,
    ptrdiff_t *info
);

/* Source: ztrsyl.f */
#define ztrsyl FORTRAN_WRAPPER(ztrsyl)
extern void ztrsyl(
    char   *trana,
    char   *tranb,
    ptrdiff_t *isgn,
    ptrdiff_t *m,
    ptrdiff_t *n,
    double *a,
    ptrdiff_t *lda,
    double *b,
    ptrdiff_t *ldb,
    double *c,
    ptrdiff_t *ldc,
    double *scale,
    ptrdiff_t *info
);

/* Source: ztrti2.f */
#define ztrti2 FORTRAN_WRAPPER(ztrti2)
extern void ztrti2(
    char   *uplo,
    char   *diag,
    ptrdiff_t *n,
    double *a,
    ptrdiff_t *lda,
    ptrdiff_t *info
);

/* Source: ztrtri.f */
#define ztrtri FORTRAN_WRAPPER(ztrtri)
extern void ztrtri(
    char   *uplo,
    char   *diag,
    ptrdiff_t *n,
    double *a,
    ptrdiff_t *lda,
    ptrdiff_t *info
);

/* Source: ztrtrs.f */
#define ztrtrs FORTRAN_WRAPPER(ztrtrs)
extern void ztrtrs(
    char   *uplo,
    char   *trans,
    char   *diag,
    ptrdiff_t *n,
    ptrdiff_t *nrhs,
    double *a,
    ptrdiff_t *lda,
    double *b,
    ptrdiff_t *ldb,
    ptrdiff_t *info
);

/* Source: ztrttf.f */
#define ztrttf FORTRAN_WRAPPER(ztrttf)
extern void ztrttf(
    char   *transr,
    char   *uplo,
    ptrdiff_t *n,
    double *a,
    ptrdiff_t *lda,
    double *arf,
    ptrdiff_t *info
);

/* Source: ztrttp.f */
#define ztrttp FORTRAN_WRAPPER(ztrttp)
extern void ztrttp(
    char   *uplo,
    ptrdiff_t *n,
    double *a,
    ptrdiff_t *lda,
    double *ap,
    ptrdiff_t *info
);

/* Source: ztzrqf.f */
#define ztzrqf FORTRAN_WRAPPER(ztzrqf)
extern void ztzrqf(
    ptrdiff_t *m,
    ptrdiff_t *n,
    double *a,
    ptrdiff_t *lda,
    double *tau,
    ptrdiff_t *info
);

/* Source: ztzrzf.f */
#define ztzrzf FORTRAN_WRAPPER(ztzrzf)
extern void ztzrzf(
    ptrdiff_t *m,
    ptrdiff_t *n,
    double *a,
    ptrdiff_t *lda,
    double *tau,
    double *work,
    ptrdiff_t *lwork,
    ptrdiff_t *info
);

/* Source: zung2l.f */
#define zung2l FORTRAN_WRAPPER(zung2l)
extern void zung2l(
    ptrdiff_t *m,
    ptrdiff_t *n,
    ptrdiff_t *k,
    double *a,
    ptrdiff_t *lda,
    double *tau,
    double *work,
    ptrdiff_t *info
);

/* Source: zung2r.f */
#define zung2r FORTRAN_WRAPPER(zung2r)
extern void zung2r(
    ptrdiff_t *m,
    ptrdiff_t *n,
    ptrdiff_t *k,
    double *a,
    ptrdiff_t *lda,
    double *tau,
    double *work,
    ptrdiff_t *info
);

/* Source: zungbr.f */
#define zungbr FORTRAN_WRAPPER(zungbr)
extern void zungbr(
    char   *vect,
    ptrdiff_t *m,
    ptrdiff_t *n,
    ptrdiff_t *k,
    double *a,
    ptrdiff_t *lda,
    double *tau,
    double *work,
    ptrdiff_t *lwork,
    ptrdiff_t *info
);

/* Source: zunghr.f */
#define zunghr FORTRAN_WRAPPER(zunghr)
extern void zunghr(
    ptrdiff_t *n,
    ptrdiff_t *ilo,
    ptrdiff_t *ihi,
    double *a,
    ptrdiff_t *lda,
    double *tau,
    double *work,
    ptrdiff_t *lwork,
    ptrdiff_t *info
);

/* Source: zungl2.f */
#define zungl2 FORTRAN_WRAPPER(zungl2)
extern void zungl2(
    ptrdiff_t *m,
    ptrdiff_t *n,
    ptrdiff_t *k,
    double *a,
    ptrdiff_t *lda,
    double *tau,
    double *work,
    ptrdiff_t *info
);

/* Source: zunglq.f */
#define zunglq FORTRAN_WRAPPER(zunglq)
extern void zunglq(
    ptrdiff_t *m,
    ptrdiff_t *n,
    ptrdiff_t *k,
    double *a,
    ptrdiff_t *lda,
    double *tau,
    double *work,
    ptrdiff_t *lwork,
    ptrdiff_t *info
);

/* Source: zungql.f */
#define zungql FORTRAN_WRAPPER(zungql)
extern void zungql(
    ptrdiff_t *m,
    ptrdiff_t *n,
    ptrdiff_t *k,
    double *a,
    ptrdiff_t *lda,
    double *tau,
    double *work,
    ptrdiff_t *lwork,
    ptrdiff_t *info
);

/* Source: zungqr.f */
#define zungqr FORTRAN_WRAPPER(zungqr)
extern void zungqr(
    ptrdiff_t *m,
    ptrdiff_t *n,
    ptrdiff_t *k,
    double *a,
    ptrdiff_t *lda,
    double *tau,
    double *work,
    ptrdiff_t *lwork,
    ptrdiff_t *info
);

/* Source: zungr2.f */
#define zungr2 FORTRAN_WRAPPER(zungr2)
extern void zungr2(
    ptrdiff_t *m,
    ptrdiff_t *n,
    ptrdiff_t *k,
    double *a,
    ptrdiff_t *lda,
    double *tau,
    double *work,
    ptrdiff_t *info
);

/* Source: zungrq.f */
#define zungrq FORTRAN_WRAPPER(zungrq)
extern void zungrq(
    ptrdiff_t *m,
    ptrdiff_t *n,
    ptrdiff_t *k,
    double *a,
    ptrdiff_t *lda,
    double *tau,
    double *work,
    ptrdiff_t *lwork,
    ptrdiff_t *info
);

/* Source: zungtr.f */
#define zungtr FORTRAN_WRAPPER(zungtr)
extern void zungtr(
    char   *uplo,
    ptrdiff_t *n,
    double *a,
    ptrdiff_t *lda,
    double *tau,
    double *work,
    ptrdiff_t *lwork,
    ptrdiff_t *info
);

/* Source: zunm2l.f */
#define zunm2l FORTRAN_WRAPPER(zunm2l)
extern void zunm2l(
    char   *side,
    char   *trans,
    ptrdiff_t *m,
    ptrdiff_t *n,
    ptrdiff_t *k,
    double *a,
    ptrdiff_t *lda,
    double *tau,
    double *c,
    ptrdiff_t *ldc,
    double *work,
    ptrdiff_t *info
);

/* Source: zunm2r.f */
#define zunm2r FORTRAN_WRAPPER(zunm2r)
extern void zunm2r(
    char   *side,
    char   *trans,
    ptrdiff_t *m,
    ptrdiff_t *n,
    ptrdiff_t *k,
    double *a,
    ptrdiff_t *lda,
    double *tau,
    double *c,
    ptrdiff_t *ldc,
    double *work,
    ptrdiff_t *info
);

/* Source: zunmbr.f */
#define zunmbr FORTRAN_WRAPPER(zunmbr)
extern void zunmbr(
    char   *vect,
    char   *side,
    char   *trans,
    ptrdiff_t *m,
    ptrdiff_t *n,
    ptrdiff_t *k,
    double *a,
    ptrdiff_t *lda,
    double *tau,
    double *c,
    ptrdiff_t *ldc,
    double *work,
    ptrdiff_t *lwork,
    ptrdiff_t *info
);

/* Source: zunmhr.f */
#define zunmhr FORTRAN_WRAPPER(zunmhr)
extern void zunmhr(
    char   *side,
    char   *trans,
    ptrdiff_t *m,
    ptrdiff_t *n,
    ptrdiff_t *ilo,
    ptrdiff_t *ihi,
    double *a,
    ptrdiff_t *lda,
    double *tau,
    double *c,
    ptrdiff_t *ldc,
    double *work,
    ptrdiff_t *lwork,
    ptrdiff_t *info
);

/* Source: zunml2.f */
#define zunml2 FORTRAN_WRAPPER(zunml2)
extern void zunml2(
    char   *side,
    char   *trans,
    ptrdiff_t *m,
    ptrdiff_t *n,
    ptrdiff_t *k,
    double *a,
    ptrdiff_t *lda,
    double *tau,
    double *c,
    ptrdiff_t *ldc,
    double *work,
    ptrdiff_t *info
);

/* Source: zunmlq.f */
#define zunmlq FORTRAN_WRAPPER(zunmlq)
extern void zunmlq(
    char   *side,
    char   *trans,
    ptrdiff_t *m,
    ptrdiff_t *n,
    ptrdiff_t *k,
    double *a,
    ptrdiff_t *lda,
    double *tau,
    double *c,
    ptrdiff_t *ldc,
    double *work,
    ptrdiff_t *lwork,
    ptrdiff_t *info
);

/* Source: zunmql.f */
#define zunmql FORTRAN_WRAPPER(zunmql)
extern void zunmql(
    char   *side,
    char   *trans,
    ptrdiff_t *m,
    ptrdiff_t *n,
    ptrdiff_t *k,
    double *a,
    ptrdiff_t *lda,
    double *tau,
    double *c,
    ptrdiff_t *ldc,
    double *work,
    ptrdiff_t *lwork,
    ptrdiff_t *info
);

/* Source: zunmqr.f */
#define zunmqr FORTRAN_WRAPPER(zunmqr)
extern void zunmqr(
    char   *side,
    char   *trans,
    ptrdiff_t *m,
    ptrdiff_t *n,
    ptrdiff_t *k,
    double *a,
    ptrdiff_t *lda,
    double *tau,
    double *c,
    ptrdiff_t *ldc,
    double *work,
    ptrdiff_t *lwork,
    ptrdiff_t *info
);

/* Source: zunmr2.f */
#define zunmr2 FORTRAN_WRAPPER(zunmr2)
extern void zunmr2(
    char   *side,
    char   *trans,
    ptrdiff_t *m,
    ptrdiff_t *n,
    ptrdiff_t *k,
    double *a,
    ptrdiff_t *lda,
    double *tau,
    double *c,
    ptrdiff_t *ldc,
    double *work,
    ptrdiff_t *info
);

/* Source: zunmr3.f */
#define zunmr3 FORTRAN_WRAPPER(zunmr3)
extern void zunmr3(
    char   *side,
    char   *trans,
    ptrdiff_t *m,
    ptrdiff_t *n,
    ptrdiff_t *k,
    ptrdiff_t *l,
    double *a,
    ptrdiff_t *lda,
    double *tau,
    double *c,
    ptrdiff_t *ldc,
    double *work,
    ptrdiff_t *info
);

/* Source: zunmrq.f */
#define zunmrq FORTRAN_WRAPPER(zunmrq)
extern void zunmrq(
    char   *side,
    char   *trans,
    ptrdiff_t *m,
    ptrdiff_t *n,
    ptrdiff_t *k,
    double *a,
    ptrdiff_t *lda,
    double *tau,
    double *c,
    ptrdiff_t *ldc,
    double *work,
    ptrdiff_t *lwork,
    ptrdiff_t *info
);

/* Source: zunmrz.f */
#define zunmrz FORTRAN_WRAPPER(zunmrz)
extern void zunmrz(
    char   *side,
    char   *trans,
    ptrdiff_t *m,
    ptrdiff_t *n,
    ptrdiff_t *k,
    ptrdiff_t *l,
    double *a,
    ptrdiff_t *lda,
    double *tau,
    double *c,
    ptrdiff_t *ldc,
    double *work,
    ptrdiff_t *lwork,
    ptrdiff_t *info
);

/* Source: zunmtr.f */
#define zunmtr FORTRAN_WRAPPER(zunmtr)
extern void zunmtr(
    char   *side,
    char   *uplo,
    char   *trans,
    ptrdiff_t *m,
    ptrdiff_t *n,
    double *a,
    ptrdiff_t *lda,
    double *tau,
    double *c,
    ptrdiff_t *ldc,
    double *work,
    ptrdiff_t *lwork,
    ptrdiff_t *info
);

/* Source: zupgtr.f */
#define zupgtr FORTRAN_WRAPPER(zupgtr)
extern void zupgtr(
    char   *uplo,
    ptrdiff_t *n,
    double *ap,
    double *tau,
    double *q,
    ptrdiff_t *ldq,
    double *work,
    ptrdiff_t *info
);

/* Source: zupmtr.f */
#define zupmtr FORTRAN_WRAPPER(zupmtr)
extern void zupmtr(
    char   *side,
    char   *uplo,
    char   *trans,
    ptrdiff_t *m,
    ptrdiff_t *n,
    double *ap,
    double *tau,
    double *c,
    ptrdiff_t *ldc,
    double *work,
    ptrdiff_t *info
);

#ifdef __cplusplus
    }   /* extern "C" */
#endif

#endif /* lapack_h */
```

### mat.h
```c
/*
 * PUBLISHed header for libmat, the MAT File library.
 *
 * Copyright 1984-2010 The MathWorks, Inc.
 * All Rights Reserved.
 */

#if defined(_MSC_VER)
# pragma once
#endif
#if defined(__GNUC__) && (__GNUC__ > 3 || (__GNUC__ == 3 && __GNUC_MINOR__ > 3))
# pragma once
#endif

#ifndef mat_published_c_api_h
#define mat_published_c_api_h

#ifndef EXTERN_C
#  ifdef __cplusplus
#    define EXTERN_C extern "C"
#  else
#    define EXTERN_C extern
#  endif
#endif

#ifndef LIBMAT_API
#  define LIBMAT_API
#endif

#include <stdio.h>  /* for FILE */

#include "matrix.h" /* for mxArray */

/* incomplete typedef for MATFile */
#ifdef __cplusplus
class MATFile;
#else
typedef struct MatFile_tag MATFile;
#endif

/*
 * Open a MAT-file "filename" using mode "mode".  Return
 * a pointer to a MATFile for use with other MAT API functions.
 *
 * Current valid entries for "mode" are
 * "r"    == read only.
 * "w"    == write only (deletes any existing file with name <filename>).
 * "w4"   == as "w", but create a MATLAB 4.0 MAT-file.
 * "w7.3" == as "w", but create a MATLAB 7.3 MAT-file.
 * "u"    == update.  Read and write allowed, existing file is not deleted.
 *
 * Return NULL if an error occurs.
 */
EXTERN_C LIBMAT_API MATFile* matOpen(const char *filename, const char * mode);

/*
 * Close a MAT-file opened with matOpen.
 * The pointer-to-MATfile argument is invalid, once matClose returns.
 * Return zero for success, EOF on error.
 */
EXTERN_C LIBMAT_API int matClose(MATFile *pMF);

/*
 * Return the ANSI C FILE pointer obtained when the MAT-file was opened.
 * Warning: the FILE pointer may be NULL in the case of a MAT file format
 * that does not allow access to the raw file pointer.
 */
EXTERN_C LIBMAT_API FILE * matGetFp(MATFile *pMF);

/*
 * Write array value with the specified name to the MAT-file, deleting any
 * previously existing variable with that name in the MAT-file.
 *
 * Return zero for success, nonzero for error.
 */
EXTERN_C LIBMAT_API int matPutVariable(MATFile * pMF, const char * name, const mxArray * pA);

/*
 * Write array value with the specified name to the MAT-file pMF, deleting any
 * previously existing variable in the MAT-file with the same name.
 *
 * The variable will be written such that when the MATLAB LOAD command
 * loads the variable, it will automatically place it in the
 * global workspace and establish a link to it in the local
 * workspace (as if the command "global <varname>" had been
 * issued after the variable was loaded.)
 *
 * Return zero for success, nonzero for error.
 */
EXTERN_C LIBMAT_API int matPutVariableAsGlobal(MATFile * pMF, const char * name, const mxArray * pA);

/*
 * Read the array value for the specified variable name from a MAT-file.
 *
 * Return NULL if an error occurs.
 */
EXTERN_C LIBMAT_API mxArray * matGetVariable(MATFile * pMF, const char * name);

/*
 * Read the next array value from the current file location of the MAT-file
 * pMF.  This function should only be used in conjunction with
 * matOpen and matClose.  Passing pMF to any other API functions
 * will cause matGetNextVariable() to work incorrectly.
 *
 * Return NULL if an error occurs.
 */
EXTERN_C LIBMAT_API mxArray * matGetNextVariable(MATFile *pMF, const char **nameptr);

/*
 * Read the array header of the next array value in a MAT-file.
 * This function should only be used in conjunction with
 * matOpen and matClose.  Passing pMF to any other API functions
 * will cause matGetNextVariableInfo to work incorrectly.
 *
 * See the description of matGetVariableInfo() for the definition
 * and valid uses of an array header.
 *
 * Return NULL if an error occurs.
 */
EXTERN_C LIBMAT_API mxArray * matGetNextVariableInfo(MATFile *pMF, const char **nameptr);

/*
 * Read the array header for the variable with the specified name from
 * the MAT-file.
 *
 * An array header contains all the same information as an
 * array, except that the pr, pi, ir, and jc data structures are
 * not allocated for non-recursive data types.  That is,
 * Cells, structures, and objects contain pointers to other
 * array headers, but numeric, string, and sparse arrays do not
 * contain valid data in their pr, pi, ir, or jc fields.
 *
 * The purpose of an array header is to gain fast access to
 * information about an array without reading all the array's
 * actual data.  Thus, functions such as mxGetM, mxGetN, and mxGetClassID
 * can be used with array headers, but mxGetPr, mxGetPi, mxGetIr, mxGetJc,
 * mxSetPr, mxSetPi, mxSetIr, and mxSetJc cannot.
 *
 * An array header should NEVER be returned to MATLAB (for example via the
 * MEX API), or any other non-matrix access API function that expects a
 * full mxArray (examples include engPutVariable(), matPutVariable(), and
 * mexPutVariable()).
 *
 * Return NULL if an error occurs.
 */
EXTERN_C LIBMAT_API mxArray * matGetVariableInfo(MATFile *pMF, const char * name);

/*
 * Remove a variable with with the specified name from the MAT-file pMF.
 *
 * Return zero on success, non-zero on error.
 */
EXTERN_C LIBMAT_API int matDeleteVariable(MATFile *pMF, const char *name);

/*
 * Get a list of the names of the arrays in a MAT-file.
 * The array of strings returned by this function contains "num"
 * entries.  It is allocated with one call to mxCalloc, and so
 * can (must) be freed with one call to mxFree.
 *
 * If there are no arrays in the MAT-file, return value
 * is NULL and num is set to zero.  If an error occurs,
 * return value is NULL and num is set to a negative number.
 */
EXTERN_C LIBMAT_API char ** matGetDir(MATFile * pMF, int *num);

#endif /* mat_published_c_api_h */
```

### matrix.h
```c
/*
 * @(#)matrix.h    generated by: makeheader 5.1.5  Tue May 24 21:08:01 2011
 *
 *		built from:	../../src/include/copyright.h
 *				../../src/include/pragma_interface.h
 *				include/published_version.h
 *				include/symver.h
 *				export/include/matrix/detail/published_fwd_decls.hpp
 *				alloccbk.cpp
 *				alloclst.cpp
 *				array.cpp
 *				array2.cpp
 *				arraycbk.cpp
 *				arraycpy.cpp
 *				assignmt.cpp
 *				bytestr.cpp
 *				catenate.cpp
 *				cellindex.cpp
 *				checkdim.cpp
 *				compat32.cpp
 *				conversions.cpp
 *				end.cpp
 *				errmsg.cpp
 *				error.cpp
 *				fmxapi.cpp
 *				fmxapi_700.cpp
 *				fmxapi_730.cpp
 *				funhdl.cpp
 *				grow.cpp
 *				ieee_wrap.cpp
 *				indexcpy.cpp
 *				iocbk.cpp
 *				marshal.cpp
 *				mcat.cpp
 *				mxarray_alloc.cpp
 *				mxassert.cpp
 *				mxequal.cpp
 *				mxuint128.cpp
 *				mxutil.cpp
 *				nameindex.cpp
 *				nargchk.cpp
 *				numconv.cpp
 *				opaque.cpp
 *				permute.cpp
 *				populate.cpp
 *				protected.cpp
 *				referenc.cpp
 *				resize.cpp
 *				rndcolon.cpp
 *				rootrecord_debug.cpp
 *				scopemgr.cpp
 *				strconv.cpp
 *				subserror.cpp
 *				transpose.cpp
 *				txtcmp.cpp
 *				undoc.cpp
 *				warning.cpp
 *				zbuffer.cpp
 *				include/compat_pub.h
 */

#if defined(_MSC_VER)
# pragma once
#endif
#if defined(__GNUC__) && (__GNUC__ > 3 || (__GNUC__ == 3 && __GNUC_MINOR__ > 3))
# pragma once
#endif

#ifndef matrix_h
#define matrix_h

/*
 * Copyright 1984-2003 The MathWorks, Inc.
 * All Rights Reserved.
 */

/* Copyright 2003-2006 The MathWorks, Inc. */

/* Only define EXTERN_C if it hasn't been defined already. This allows
 * individual modules to have more control over managing their exports.
 */
#ifndef EXTERN_C

#ifdef __cplusplus
  #define EXTERN_C extern "C"
#else
  #define EXTERN_C extern
#endif

#endif

/* Version 7.4.0 */
#define MX_API_VER 0x07040000

#ifndef matrix_symver_h

/*
 * PUBLISHED APIs with changes in MATLAB 7.3
 */

#if !defined(MX_COMPAT_32) || defined(MX_INTERNAL_730)

/*
 * Include this uniformly on non-Linux platforms (no .symver)
 * Include it only internal to the matrix library on Linux
 */
#if !defined(__linux__) || defined(MX_INTERNAL_730)

#ifndef mxSetProperty
# define mxSetProperty mxSetProperty_730
#endif

#ifndef mxGetProperty
# define mxGetProperty mxGetProperty_730
#endif

#ifndef mxSetField
# define mxSetField mxSetField_730
#endif

#ifndef mxSetFieldByNumber
# define mxSetFieldByNumber mxSetFieldByNumber_730
#endif

#ifndef mxGetFieldByNumber
# define mxGetFieldByNumber mxGetFieldByNumber_730
#endif

#ifndef mxGetField
# define mxGetField mxGetField_730
#endif

#ifndef mxCreateStructMatrix
# define mxCreateStructMatrix mxCreateStructMatrix_730
#endif

#ifndef mxCreateCellMatrix
# define mxCreateCellMatrix mxCreateCellMatrix_730
#endif

#ifndef mxCreateCharMatrixFromStrings
# define mxCreateCharMatrixFromStrings mxCreateCharMatrixFromStrings_730
#endif

#ifndef mxGetString
# define mxGetString mxGetString_730
#endif

#ifndef mxGetNumberOfDimensions
# define mxGetNumberOfDimensions mxGetNumberOfDimensions_730
#endif

#ifndef mxGetDimensions
# define mxGetDimensions mxGetDimensions_730
#endif

#ifndef mxSetDimensions
# define mxSetDimensions mxSetDimensions_730
#endif

#ifndef mxSetIr
# define mxSetIr mxSetIr_730
#endif

#ifndef mxGetIr
# define mxGetIr mxGetIr_730
#endif

#ifndef mxSetJc
# define mxSetJc mxSetJc_730
#endif

#ifndef mxGetJc
# define mxGetJc mxGetJc_730
#endif

#ifndef mxCreateStructArray
# define mxCreateStructArray mxCreateStructArray_730
#endif

#ifndef mxCreateCharArray
# define mxCreateCharArray mxCreateCharArray_730
#endif

#ifndef mxCreateNumericArray
# define mxCreateNumericArray mxCreateNumericArray_730
#endif

#ifndef mxCreateCellArray
# define mxCreateCellArray mxCreateCellArray_730
#endif

#ifndef mxCreateLogicalArray
# define mxCreateLogicalArray mxCreateLogicalArray_730
#endif

#ifndef mxGetCell
# define mxGetCell mxGetCell_730
#endif

#ifndef mxSetCell
# define mxSetCell mxSetCell_730
#endif

#ifndef mxSetNzmax
# define mxSetNzmax mxSetNzmax_730
#endif

#ifndef mxSetN
# define mxSetN mxSetN_730
#endif

#ifndef mxSetM
# define mxSetM mxSetM_730
#endif

#ifndef mxGetNzmax
# define mxGetNzmax mxGetNzmax_730
#endif

#ifndef mxCreateDoubleMatrix
# define mxCreateDoubleMatrix mxCreateDoubleMatrix_730
#endif

#ifndef mxCreateNumericMatrix
# define mxCreateNumericMatrix mxCreateNumericMatrix_730
#endif

#ifndef mxCreateLogicalMatrix
# define mxCreateLogicalMatrix mxCreateLogicalMatrix_730
#endif

#ifndef mxCreateSparse
# define mxCreateSparse mxCreateSparse_730
#endif

#ifndef mxCreateSparseLogicalMatrix
# define mxCreateSparseLogicalMatrix mxCreateSparseLogicalMatrix_730
#endif

#ifndef mxGetNChars
# define mxGetNChars mxGetNChars_730
#endif

#ifndef mxCreateStringFromNChars
# define mxCreateStringFromNChars mxCreateStringFromNChars_730
#endif

#ifndef mxCalcSingleSubscript
# define mxCalcSingleSubscript mxCalcSingleSubscript_730
#endif

#ifndef mxGetDimensions_fcn
# define mxGetDimensions_fcn mxGetDimensions_730
#endif

#else

#ifndef mxGetDimensions_fcn
# define mxGetDimensions_fcn mxGetDimensions
#endif

#endif /* !__linux__ || MX_INTERNAL_730 */

#else

#ifndef mxGetDimensions_fcn
# define mxGetDimensions_fcn mxGetDimensions_700
#endif

#endif /* !MX_COMPAT_32 || MX_INTERNAL_730 */

#endif /* matrix_symver_h */

/* Copyright 2008-2010 The MathWorks, Inc. */

/*
 * NOTE: The contents of this header are ultimately PUBLISHED in
 * extern/include/matrix.h.
 */

#ifndef MATHWORKS_MATRIX_DETAIL_PUBLISHED_FWD_DECLS_HPP
#define MATHWORKS_MATRIX_DETAIL_PUBLISHED_FWD_DECLS_HPP

#include <stddef.h>
#include <tmwtypes.h>

/**
 * Forward declaration for mxArray
 */
typedef struct mxArray_tag mxArray;

/**
 * Type representing the signature for MEX functions.
 */
typedef void (*mxFunctionPtr) (int nlhs, mxArray *plhs[], int nrhs, mxArray *prhs[]);

/**
 * Maximum mxArray name length
 */
#define mxMAXNAM TMW_NAME_LENGTH_MAX

/**
 * Logical type
 */
typedef bool mxLogical;

/**
 * Typedef required for Unicode support in MATLAB
 */
typedef CHAR16_T mxChar;

/**
 * Enumeration corresponding to all the valid mxArray types.
 */
typedef enum
{
    mxUNKNOWN_CLASS = 0,
    mxCELL_CLASS,
    mxSTRUCT_CLASS,
    mxLOGICAL_CLASS,
    mxCHAR_CLASS,
    mxVOID_CLASS,
    mxDOUBLE_CLASS,
    mxSINGLE_CLASS,
    mxINT8_CLASS,
    mxUINT8_CLASS,
    mxINT16_CLASS,
    mxUINT16_CLASS,
    mxINT32_CLASS,
    mxUINT32_CLASS,
    mxINT64_CLASS,
    mxUINT64_CLASS,
    mxFUNCTION_CLASS,
    mxOPAQUE_CLASS,
    mxOBJECT_CLASS, /* keep the last real item in the list */
#if defined(_LP64) || defined(_WIN64)
    mxINDEX_CLASS = mxUINT64_CLASS,
#else
    mxINDEX_CLASS = mxUINT32_CLASS,
#endif
    /* TEMPORARY AND NASTY HACK UNTIL mxSPARSE_CLASS IS COMPLETELY ELIMINATED */
    mxSPARSE_CLASS = mxVOID_CLASS /* OBSOLETE! DO NOT USE */
}
mxClassID;

/**
 * Indicates whether floating-point mxArrays are real or complex.
 */
typedef enum
{
    mxREAL,
    mxCOMPLEX
}
mxComplexity;

#endif /* MATHWORKS_MATRIX_DETAIL_PUBLISHED_FWD_DECLS_HPP */

#include <stddef.h>	/* size_t */

/*
 * allocate memory, notifying registered listener
 */
EXTERN_C void *mxMalloc(
    size_t	n		/* number of bytes */
    );

/*
 * allocate cleared memory, notifying registered listener.
 */
EXTERN_C void *mxCalloc(
    size_t	n,	/* number of objects */
    size_t	size	/* size of objects */
    );

/*
 * free memory, notifying registered listener.
 */
EXTERN_C void mxFree(void *ptr)	/* pointer to memory to be freed */;

/*
 * reallocate memory, notifying registered listener.
 */
EXTERN_C void *mxRealloc(void *ptr, size_t size);

/*
 * Return the class (catergory) of data that the array holds.
 */
EXTERN_C mxClassID mxGetClassID(const mxArray *pa);

/*
 * Get pointer to data
 */
EXTERN_C void *mxGetData(
    const mxArray *pa		/* pointer to array */
    );

/*
 * Set pointer to data
 */
EXTERN_C void mxSetData(
    mxArray *pa,		/* pointer to array */
    void  *newdata		/* pointer to data */
    );

/*
 * Determine whether the specified array contains numeric (as opposed
 * to cell or struct) data.
 */
EXTERN_C bool mxIsNumeric(const mxArray *pa);

/*
 * Determine whether the given array is a cell array.
 */
EXTERN_C bool mxIsCell(const mxArray *pa);

/*
 * Determine whether the given array's logical flag is on.
 */
EXTERN_C bool mxIsLogical(const mxArray *pa);

/*
 * Determine whether the given array contains character data.
 */
EXTERN_C bool mxIsChar(const mxArray *pa);

/*
 * Determine whether the given array is a structure array.
 */
EXTERN_C bool mxIsStruct(const mxArray *pa);

/*
 * Determine whether the given array is an opaque array.
 */
EXTERN_C bool mxIsOpaque(const mxArray *pa);

/*
 * Returns true if specified array is a function object.
 */
EXTERN_C bool mxIsFunctionHandle(const mxArray *pa);

/*
 * This function is deprecated and is preserved only for backward compatibility.
 * DO NOT USE if possible.
 * Is array user defined MATLAB v5 object
 */
EXTERN_C bool mxIsObject(
    const mxArray *pa		/* pointer to array */
    );

/*
 * Get imaginary data pointer for numeric array
 */
EXTERN_C void *mxGetImagData(
    const mxArray *pa		/* pointer to array */
    );

/*
 * Set imaginary data pointer for numeric array
 */
EXTERN_C void mxSetImagData(
    mxArray *pa,		/* pointer to array */
    void    *newdata		/* imaginary data array pointer */
    );

/*
 * Determine whether the given array contains complex data.
 */
EXTERN_C bool mxIsComplex(const mxArray *pa);

/*
 * Determine whether the given array is a sparse (as opposed to full).
 */
EXTERN_C bool mxIsSparse(const mxArray *pa);

/*
 * Determine whether the specified array represents its data as
 * double-precision floating-point numbers.
 */
EXTERN_C bool mxIsDouble(const mxArray *pa);

/*
 * Determine whether the specified array represents its data as
 * single-precision floating-point numbers.
 */
EXTERN_C bool mxIsSingle(const mxArray *pa);

/*
 * Determine whether the specified array represents its data as
 * signed 8-bit integers.
 */
EXTERN_C bool mxIsInt8(const mxArray *pa);

/*
 * Determine whether the specified array represents its data as
 * unsigned 8-bit integers.
 */
EXTERN_C bool mxIsUint8(const mxArray *pa);

/*
 * Determine whether the specified array represents its data as
 * signed 16-bit integers.
 */
EXTERN_C bool mxIsInt16(const mxArray *pa);

/*
 * Determine whether the specified array represents its data as
 * unsigned 16-bit integers.
 */
EXTERN_C bool mxIsUint16(const mxArray *pa);

/*
 * Determine whether the specified array represents its data as
 * signed 32-bit integers.
 */
EXTERN_C bool mxIsInt32(const mxArray *pa);

/*
 * Determine whether the specified array represents its data as
 * unsigned 32-bit integers.
 */
EXTERN_C bool mxIsUint32(const mxArray *pa);

/*
 * Determine whether the specified array represents its data as
 * signed 64-bit integers.
 */
EXTERN_C bool mxIsInt64(const mxArray *pa);

/*
 * Determine whether the specified array represents its data as
 * unsigned 64-bit integers.
 */
EXTERN_C bool mxIsUint64(const mxArray *pa);

/*
 * Get number of dimensions in array
 */
EXTERN_C mwSize mxGetNumberOfDimensions(const mxArray *pa);

/*
 * Get pointer to dimension array
 */
EXTERN_C const mwSize *mxGetDimensions(const mxArray *pa);

/*
 * Get number of elements in array
 */
EXTERN_C size_t mxGetNumberOfElements(
    const mxArray *pa		/* pointer to array */
    );

/*
 * Get real data pointer for numeric array
 */
EXTERN_C double *mxGetPr(
    const mxArray *pa		/* pointer to array */
    );

/*
 * Set real data pointer for numeric array
 */
EXTERN_C void mxSetPr(
    mxArray *pa,		/* pointer to array */
    double  *pr			/* real data array pointer */
    );

/*
 * Get imaginary data pointer for numeric array
 */
EXTERN_C double *mxGetPi(
    const mxArray *pa		/* pointer to array */
    );

/*
 * Set imaginary data pointer for numeric array
 */
EXTERN_C void mxSetPi(
    mxArray *pa,		/* pointer to array */
    double  *pi			/* imaginary data array pointer */
    );

/*
 * Get string array data
 */
EXTERN_C mxChar *mxGetChars(
    const mxArray *pa		/* pointer to array */
    );

/*
 * Get 8 bits of user data stored in the mxArray header.  NOTE: This state
 * of these bits are not guaranteed to be preserved after API function
 * calls.
 */
EXTERN_C int mxGetUserBits(
    const mxArray	*pa		/* pointer to array */
    );

/*
 * Set 8 bits of user data stored in the mxArray header. NOTE: This state
 * of these bits are not guaranteed to be preserved after API function
 * calls.
 */
EXTERN_C void mxSetUserBits(
	mxArray	*pa,		/* pointer to array */
	int	value
    );

/*
 * Get the real component of the specified array's first data element.
 */
EXTERN_C double mxGetScalar(const mxArray *pa);

/*
 * Inform Watcom compilers that scalar double return values
 * will be in the FPU register.
 */
#ifdef __WATCOMC__
#pragma aux mxGetScalar value [8087];
#endif

/*
 * Is the isFromGlobalWorkspace bit set?
 */
EXTERN_C bool mxIsFromGlobalWS(const mxArray *pa);

/*
 * Set the isFromGlobalWorkspace bit.
 */
EXTERN_C void mxSetFromGlobalWS(mxArray *pa, bool global);

/*
 * Get row dimension
 */
EXTERN_C size_t mxGetM(const mxArray *pa);

/*
 * Set row dimension
 */
EXTERN_C void mxSetM(mxArray *pa, mwSize m);

/*
 * Get column dimension
 */
EXTERN_C size_t mxGetN(const mxArray *pa);

/*
 * Is array empty
 */
EXTERN_C bool mxIsEmpty(
    const mxArray *pa		/* pointer to array */
    );

/*
 * Get row data pointer for sparse numeric array
 */
EXTERN_C mwIndex *mxGetIr(const mxArray *pa);

/*
 * Set row data pointer for numeric array
 */
EXTERN_C void mxSetIr(mxArray *pa, mwIndex *newir);

/*
 * Get column data pointer for sparse numeric array
 */
EXTERN_C mwIndex *mxGetJc(const mxArray *pa);

/*
 * Set column data pointer for numeric array
 */
EXTERN_C void mxSetJc(mxArray *pa, mwIndex *newjc);

/*
 * Get maximum nonzero elements for sparse numeric array
 */
EXTERN_C mwSize mxGetNzmax(const mxArray *pa);

/*
 * Set maximum nonzero elements for numeric array
 */
EXTERN_C void mxSetNzmax(mxArray *pa, mwSize nzmax);

/*
 * Get array data element size
 */
EXTERN_C size_t mxGetElementSize(const mxArray *pa);

/*
 * Return the offset (in number of elements) from the beginning of
 * the array to a given subscript.
 */
EXTERN_C mwIndex mxCalcSingleSubscript(const mxArray *pa, mwSize nsubs, const mwIndex *subs);

/*
 * Get number of structure fields in array
 * Returns 0 if mxArray is non-struct.
 */
EXTERN_C int mxGetNumberOfFields(
    const mxArray *pa		/* pointer to array */
    );

/*
 * Get a pointer to the specified cell element.
 */
EXTERN_C mxArray *mxGetCell(const mxArray *pa, mwIndex i);

/*
 * Set an element in a cell array to the specified value.
 */
EXTERN_C void mxSetCell(mxArray *pa, mwIndex i, mxArray *value);

/*
 * Return pointer to the nth field name
 */
EXTERN_C const char *mxGetFieldNameByNumber(const mxArray *pa, int n);

/*
 * Get the index to the named field.
 */
EXTERN_C int mxGetFieldNumber(const mxArray *pa, const char *name);

/*
 * Return a pointer to the contents of the named field for
 * the ith element (zero based).
 */
EXTERN_C mxArray *mxGetFieldByNumber(const mxArray *pa, mwIndex i, int fieldnum);

/*
 * Set pa[i][fieldnum] = value
 */
EXTERN_C void mxSetFieldByNumber(mxArray *pa, mwIndex i, int fieldnum, mxArray *value);

/*
 * Return a pointer to the contents of the named field for the ith
 * element (zero based).  Returns NULL on no such field or if the
 * field itself is NULL
 */
EXTERN_C mxArray *mxGetField(const mxArray *pa, mwIndex i, const char *fieldname);

/*
 * Sets the contents of the named field for the ith element (zero based).
 * The input 'value' is stored in the input array 'pa' - no copy is made.
 */
EXTERN_C void mxSetField(mxArray *pa, mwIndex i, const char *fieldname, mxArray *value);

/*
 * mxGetProperty returns the value of a property for a given object and index.
 * The property must be public.
 *
 * If the given property name doesn't exist, isn't public, or the object isn't
 * the right type, then mxGetProperty returns NULL.
 */
EXTERN_C mxArray *mxGetProperty(const mxArray *pa, const mwIndex i, const char *propname);

/*
 * mxSetProperty sets the value of a property for a given object and index.
 * The property must be public.
 *
 */
EXTERN_C void mxSetProperty(mxArray *pa, mwIndex i, const char *propname, const mxArray *value);

/*
 * Return the name of an array's class.
 */
EXTERN_C const char *mxGetClassName(const mxArray *pa);

/*
 * Determine whether an array is a member of the specified class.
 */
EXTERN_C bool mxIsClass(const mxArray *pa, const char *name);

#include <stdlib.h>

#if !defined(MX_COMPAT_32) || defined(MX_INTERNAL_730)

/*
 * Create a numeric matrix and initialize all its data elements to 0.
 */
EXTERN_C mxArray *mxCreateNumericMatrix(mwSize m, mwSize n, mxClassID classid, mxComplexity flag);

#endif

/*
 * Set column dimension
 */
EXTERN_C void mxSetN(mxArray *pa, mwSize n);

/*
 * Set dimension array and number of dimensions.  Returns 0 on success and 1
 * if there was not enough memory available to reallocate the dimensions array.
 */
EXTERN_C int mxSetDimensions(mxArray *pa, const mwSize *size, mwSize ndims);

/*
 * mxArray destructor
 */
EXTERN_C void mxDestroyArray(mxArray *pa);

/*
 * Create a numeric array and initialize all its data elements to 0.
 *
 * Similar to mxCreateNumericMatrix, in a standalone application,
 * out-of-memory will mean a NULL pointer is returned.
 */
EXTERN_C mxArray *mxCreateNumericArray(mwSize ndim, const mwSize *dims, mxClassID classid, mxComplexity flag);

/*
 * Create an N-Dimensional array to hold string data;
 * initialize all elements to 0.
 */
EXTERN_C mxArray *mxCreateCharArray(mwSize ndim, const mwSize *dims);

/*
 * Create a two-dimensional array to hold double-precision
 * floating-point data; initialize each data element to 0.
 */
EXTERN_C mxArray *mxCreateDoubleMatrix(mwSize m, mwSize n, mxComplexity flag);

/*
 * Get a properly typed pointer to the elements of a logical array.
 */
EXTERN_C mxLogical *mxGetLogicals(const mxArray *pa);

/*
 * Create a logical array and initialize its data elements to false.
 */
EXTERN_C mxArray *mxCreateLogicalArray(mwSize ndim, const mwSize *dims);

#if !defined(MX_COMPAT_32) || defined(MX_INTERNAL_730)

/*
 * Create a two-dimensional array to hold logical data and
 * initializes each data element to false.
 */
EXTERN_C mxArray *mxCreateLogicalMatrix(mwSize m, mwSize n);

#endif

/*
 * Create a logical scalar mxArray having the specified value.
 */
EXTERN_C mxArray *mxCreateLogicalScalar(bool value);

/*
 * Returns true if we have a valid logical scalar mxArray.
 */
EXTERN_C bool mxIsLogicalScalar(const mxArray *pa);

/*
 * Returns true if the logical scalar value is true.
 */
EXTERN_C bool mxIsLogicalScalarTrue(const mxArray *pa);

/*
 * Create a double-precision scalar mxArray initialized to the
 * value specified
 */
EXTERN_C mxArray *mxCreateDoubleScalar(double value);

/*
 * Create a 2-Dimensional sparse array.
 */
EXTERN_C mxArray *mxCreateSparse(mwSize m, mwSize n, mwSize nzmax, mxComplexity flag);

/*
 * Create a 2-D sparse logical array
 */
EXTERN_C mxArray *mxCreateSparseLogicalMatrix(mwSize m, mwSize n, mwSize nzmax);

/*
 * Copies characters from a MATLAB array to a char array
 * This function will attempt to perform null termination if it is possible.
 * nChars is the number of bytes in the output buffer
 */
EXTERN_C void mxGetNChars(const mxArray *pa, char *buf, mwSize nChars);

/*
 * Converts a string array to a C-style string. The C-style string is in the
 * local codepage encoding. If the conversion for the entire Unicode string
 * cannot fit into the supplied character buffer, then the conversion includes
 * the last whole codepoint that will fit into the buffer. The string is thus
 * truncated at the greatest possible whole codepoint and does not split code-
 * points.
 */
EXTERN_C int mxGetString(const mxArray *pa, char *buf, mwSize buflen);

/*
 * Create a NULL terminated C string from an mxArray of type mxCHAR_CLASS
 * Supports multibyte character sets.  The resulting string must be freed
 * with mxFree.  Returns NULL on out of memory or non-character arrays.
 */
EXTERN_C char *mxArrayToString(const mxArray *pa);

/*
 * Create a 1-by-n string array initialized to str. The supplied string is
 * presumed to be in the local codepage encoding. The character data format
 * in the mxArray will be UTF-16.
 */
EXTERN_C mxArray *mxCreateStringFromNChars(const char *str, mwSize n);

/*
 * Create a 1-by-n string array initialized to null terminated string
 * where n is the length of the string.
 */
EXTERN_C mxArray *mxCreateString(const char *str);

/*
 * Create a string array initialized to the strings in str.
 */
EXTERN_C mxArray *mxCreateCharMatrixFromStrings(mwSize m, const char **str);

/*
 * Create a 2-Dimensional cell array, with each cell initialized
 * to NULL.
 */
EXTERN_C mxArray *mxCreateCellMatrix(mwSize m, mwSize n);

/*
 * Create an N-Dimensional cell array, with each cell initialized
 * to NULL.
 */
EXTERN_C mxArray *mxCreateCellArray(mwSize ndim, const mwSize *dims);

/*
 * Create a 2-Dimensional structure array having the specified fields;
 * initialize all values to NULL.
 */
EXTERN_C mxArray *mxCreateStructMatrix(size_t m, size_t n, int nfields, const char **fieldnames);

/*
 * Create an N-Dimensional structure array having the specified fields;
 * initialize all values to NULL.
 */
EXTERN_C mxArray *mxCreateStructArray(mwSize ndim, const mwSize *dims, int nfields,
								const char **fieldnames);

/*
 * Make a deep copy of an array, return a pointer to the copy.
 */
EXTERN_C mxArray *mxDuplicateArray(const mxArray *in);

/*
 * Set classname of an unvalidated object array.  It is illegal to
 * call this function on a previously validated object array.
 * Return 0 for success, 1 for failure.
 */
EXTERN_C int mxSetClassName(mxArray *pa, const char *classname);

/*
 * Add a field to a structure array. Returns field number on success or -1
 * if inputs are invalid or an out of memory condition occurs.
 */
EXTERN_C int mxAddField(mxArray *pa, const char *fieldname);

/*
 * Remove a field from a structure array.  Does nothing if no such field exists.
 * Does not destroy the field itself.
*/
EXTERN_C void mxRemoveField(mxArray *pa, int field);

/*
 * Function for obtaining MATLAB's concept of EPS
 */
EXTERN_C double mxGetEps(void);

/*
 * Function for obtaining MATLAB's concept of INF (Used in MEX-File callback).
 */
EXTERN_C double mxGetInf(void);

/*
 * Function for obtaining MATLAB's concept of NaN (Used in MEX-File callback).
 */
EXTERN_C double mxGetNaN(void);

/*
 * Inform Watcom compilers that scalar double return values
 * will be in the FPU register.
 */
#ifdef __WATCOMC__
#pragma aux mxGetEps value [8087];
#pragma aux mxGetInf value [8087];
#pragma aux mxGetNaN value [8087];
#endif

/*
 * test for finiteness in a machine-independent manner
 */
EXTERN_C bool mxIsFinite(
    double x                  /* value to test */
    );

/*
 * test for infinity in a machine-independent manner
 */
EXTERN_C bool mxIsInf(
    double x                  /* value to test */
    );

/*
 * test for NaN in a machine-independent manner
 */
EXTERN_C bool mxIsNaN(
    double x                  /* value to test */
    );

/*
mxAssert(int expression, char *error_message)
---------------------------------------------

  Similar to ANSI C's assert() macro, the mxAssert macro checks the
  value of an assertion, continuing execution only if the assertion
  holds.  If 'expression' evaluates to be true, then the mxAssert does
  nothing.  If, however, 'expression' is false, then mxAssert prints an
  error message to the MATLAB Command Window, consisting of the failed
  assertion's expression, the file name and line number where the failed
  assertion occurred, and the string 'error_message'.  'error_message'
  allows the user to specify a more understandable description of why
  the assertion failed.  (Use an empty string if no extra description
  should follow the failed assertion message.)  After a failed
  assertion, control returns to the MATLAB command line.

  mxAssertS, (the S for Simple), takes the same inputs as mxAssert.  It
  does not print the text of the failed assertion, only the file and
  line where the assertion failed, and the explanatory error_message.

  Note that script MEX will turn off these assertions when building
  optimized MEX-functions, so they should be used for debugging
  purposes only.
*/

#ifdef MATLAB_MEX_FILE
#  ifndef NDEBUG

EXTERN_C void mexPrintAssertion(const char *test,
		       const char *fname,
		       int linenum,
		       const char *message);

#    define mxAssert(test, message) ( (test) ? (void) 0 : mexPrintAssertion(": " #test ",", __FILE__, __LINE__, message))
#    define mxAssertS(test, message) ( (test) ? (void) 0 : mexPrintAssertion("", __FILE__, __LINE__, message))
#  else
#    define mxAssert(test, message) ((void) 0)
#    define mxAssertS(test, message) ((void) 0)
#  endif
#else
#  include <assert.h>
#  define mxAssert(test, message) assert(test)
#  define mxAssertS(test, message) assert(test)
#endif

#include <stdlib.h>

#ifdef MX_COMPAT_32
/*
 * 32-bit compatibility APIs
 */

#ifdef __cplusplus
extern "C" {
#endif

/* Cannot inline these one on 64-bit platforms */
#if defined(_LP64) || defined(_WIN64)
#undef mxGetDimensions
#undef mxSetDimensions
#undef mxSetIr
#undef mxGetIr
#undef mxSetJc
#undef mxGetJc
#undef mxCreateStructArray
#undef mxCreateCharArray
#undef mxCreateNumericArray
#undef mxCreateCellArray
#undef mxCreateLogicalArray
#undef mxGetM
#undef mxCalcSingleSubscript
#endif

#ifndef mxSetProperty
#define mxSetProperty mxSetProperty_700
#endif
void mxSetProperty_700(mxArray *, int, const char *, const mxArray *);

#ifndef mxGetProperty
#define mxGetProperty mxGetProperty_700
#endif
mxArray *mxGetProperty_700(const mxArray *, int, const char *);

#ifndef mxSetField
#define mxSetField mxSetField_700
#endif
void mxSetField_700(mxArray *, int, const char *, mxArray *);

#ifndef mxSetFieldByNumber
#define mxSetFieldByNumber mxSetFieldByNumber_700
#endif
void mxSetFieldByNumber_700(mxArray *, int, int, mxArray *);

#ifndef mxGetFieldByNumber
#define mxGetFieldByNumber mxGetFieldByNumber_700
#endif
mxArray *mxGetFieldByNumber_700(const mxArray *, int, int);

#ifndef mxGetField
#define mxGetField mxGetField_700
#endif
mxArray *mxGetField_700(const mxArray *, int, const char *);

#ifndef mxCreateStructMatrix
#define mxCreateStructMatrix mxCreateStructMatrix_700
#endif
mxArray *mxCreateStructMatrix_700(int, int, int, const char **);

#ifndef mxCreateCellMatrix
#define mxCreateCellMatrix mxCreateCellMatrix_700
#endif
mxArray *mxCreateCellMatrix_700(int, int);

#ifndef mxCreateCharMatrixFromStrings
#define mxCreateCharMatrixFromStrings mxCreateCharMatrixFromStrings_700
#endif
mxArray *mxCreateCharMatrixFromStrings_700(int, const char **);

#ifndef mxGetString
#define mxGetString mxGetString_700
#endif
int mxGetString_700(const mxArray *, char *, int);

#ifndef mxGetNumberOfDimensions
#define mxGetNumberOfDimensions mxGetNumberOfDimensions_700
#endif
int mxGetNumberOfDimensions_700(const mxArray *);

#ifndef mxGetDimensions
#define mxGetDimensions mxGetDimensions_700
#endif
const int *mxGetDimensions_700(const mxArray *);

#ifndef mxSetDimensions
#define mxSetDimensions mxSetDimensions_700
#endif
int mxSetDimensions_700(mxArray *, const int *, int);

#ifndef mxSetIr
#define mxSetIr mxSetIr_700
#endif
void mxSetIr_700(mxArray *, int *);

#ifndef mxGetIr
#define mxGetIr mxGetIr_700
#endif
int *mxGetIr_700(const mxArray *);

#ifndef mxSetJc
#define mxSetJc mxSetJc_700
#endif
void mxSetJc_700(mxArray *, int *);

#ifndef mxGetJc
#define mxGetJc mxGetJc_700
#endif
int *mxGetJc_700(const mxArray *);

#ifndef mxCreateStructArray
#define mxCreateStructArray mxCreateStructArray_700
#endif
mxArray *mxCreateStructArray_700(int, const int *, int, const char **);

#ifndef mxCreateCharArray
#define mxCreateCharArray mxCreateCharArray_700
#endif
mxArray *mxCreateCharArray_700(int, const int *);

#ifndef mxCreateNumericArray
#define mxCreateNumericArray mxCreateNumericArray_700
#endif
mxArray *mxCreateNumericArray_700(int, const int *, mxClassID, mxComplexity);

#ifndef mxCreateCellArray
#define mxCreateCellArray mxCreateCellArray_700
#endif
mxArray *mxCreateCellArray_700(int, const int *);

#ifndef mxCreateLogicalArray
#define mxCreateLogicalArray mxCreateLogicalArray_700
#endif
mxArray *mxCreateLogicalArray_700(int, const int *);

#ifndef mxGetCell
#define mxGetCell mxGetCell_700
#endif
mxArray *mxGetCell_700(const mxArray *, int);

#ifndef mxSetCell
#define mxSetCell mxSetCell_700
#endif
void mxSetCell_700(mxArray *, int, mxArray *);

#ifndef mxSetNzmax
#define mxSetNzmax mxSetNzmax_700
#endif
void mxSetNzmax_700(mxArray *, int);

#ifndef mxSetN
#define mxSetN mxSetN_700
#endif
void mxSetN_700(mxArray *, int);

#ifndef mxSetM
#define mxSetM mxSetM_700
#endif
void mxSetM_700(mxArray *, int);

#ifndef mxGetNzmax
#define mxGetNzmax mxGetNzmax_700
#endif
int mxGetNzmax_700(const mxArray *);

#ifndef mxCreateDoubleMatrix
#define mxCreateDoubleMatrix mxCreateDoubleMatrix_700
#endif
mxArray *mxCreateDoubleMatrix_700(int, int, mxComplexity);

#ifndef mxCreateNumericMatrix
#define mxCreateNumericMatrix mxCreateNumericMatrix_700
#endif
mxArray *mxCreateNumericMatrix_700(int, int, mxClassID, int);

#ifndef mxCreateLogicalMatrix
#define mxCreateLogicalMatrix mxCreateLogicalMatrix_700
#endif
mxArray *mxCreateLogicalMatrix_700(unsigned int, unsigned int);

#ifndef mxCreateSparse
#define mxCreateSparse mxCreateSparse_700
#endif
mxArray *mxCreateSparse_700(int, int, int, mxComplexity);

#ifndef mxCreateSparseLogicalMatrix
#define mxCreateSparseLogicalMatrix mxCreateSparseLogicalMatrix_700
#endif
mxArray *mxCreateSparseLogicalMatrix_700(int, int, int);

#ifndef mxGetNChars
#define mxGetNChars mxGetNChars_700
#endif
void mxGetNChars_700(const mxArray *, char *, int);

#ifndef mxCreateStringFromNChars
#define mxCreateStringFromNChars mxCreateStringFromNChars_700
#endif
mxArray *mxCreateStringFromNChars_700(const char *, int);

#ifndef mxCalcSingleSubscript
#define mxCalcSingleSubscript mxCalcSingleSubscript_700
#endif
int mxCalcSingleSubscript_700(const mxArray *, int, const int *);

#ifdef __cplusplus
}
#endif

#endif /* #ifdef MX_COMPAT_32 */

#endif /* matrix_h */
```

### mdl_info.h
```c
/*
 * Copyright 1994-2002 The MathWorks, Inc.
 *
 * File: mdl_info.h     $Revision: 1.9 $
 *
 * Abstract:
 *   Model tuning information.  Use the provided structure access methods
 *   whenever possible.
 *
 *   For details about these structures see MATLAB/rtw/c/src/pt_readme.txt
 *   and the Real-Time Workshop User's guide.
 */

#ifndef __MDL_INFO__
#define __MDL_INFO__

#include <tmwtypes.h>
#include <pt_info.h>
#include <bio_sig.h>

typedef struct ModelMappingInfo_tag {
  /* block signal monitoring */
  struct {
    BlockIOSignals const *blockIOSignals;    /* Block signals map             */
    uint_T               numBlockIOSignals;  /* Num signals in map            */
  } Signals;

  /* parameter tuning */
  struct {
    BlockTuning const    *blockTuning;       /* Block parameters map          */
    VariableTuning const *variableTuning;    /* Variable parameters map       */
    void * const         *parametersMap;     /* Parameter index map           */
    uint_T const         *dimensionsMap;     /* Dimensions index map          */
    uint_T                numBlockTuning;    /* Num block parameters in map   */
    uint_T                numVariableTuning; /* Num variable parameter in map */
  } Parameters;
} ModelMappingInfo;

#define mmiGetBlockIOSignals(MMI)    (MMI)->Signals.blockIOSignals
#define mmiGetNumBlockIOSignals(MMI) (MMI)->Signals.numBlockIOSignals

#define mmiGetBlockTuning(MMI)       (MMI)->Parameters.blockTuning
#define mmiGetVariableTuning(MMI)    (MMI)->Parameters.variableTuning
#define mmiGetParametersMap(MMI)     (MMI)->Parameters.parametersMap
#define mmiGetDimensionsMap(MMI)     (MMI)->Parameters.dimensionsMap
#define mmiGetNumBlockParams(MMI)    (MMI)->Parameters.numBlockTuning
#define mmiGetNumVariableParams(MMI) (MMI)->Parameters.numVariableTuning

#define mmiGetBlockTuningBlockName(MMI,i)  (MMI)->Parameters.blockTuning[i].blockName
#define mmiGetBlockTuningParamName(MMI,i)  (MMI)->Parameters.blockTuning[i].paramName
#define mmiGetBlockTuningParamInfo(MMI,i)  (&((MMI)->Parameters.blockTuning[i].ptRec))

#define mmiGetVariableTuningVarName(MMI,i) (MMI)->Parameters.variableTuning[i].varName
#define mmiGetVariableTuningVarInfo(MMI,i) (&((MMI)->Parameters.variableTuning[i].ptRec))

#endif  /* __MDL_INFO__ */
```

### mem_mgr.h
```c
/*
 * Copyright 1994-2002 The MathWorks, Inc.
 *
 * File: mem_mgr.h     $Revision: 1.1.6.1 $
 *
 * Abstract:
 */

#ifndef __MEM_MGR__
#define __MEM_MGR__

struct MemBufHdr {
    struct MemBufHdr *memBufNext;
    struct MemBufHdr *memBufPrev;
    char   *MemBuf;
    int    size;
};

typedef struct MemBufHdr MemBufHdr;

extern void ExtModeFree(void *mem);

extern void *ExtModeMalloc(uint32_T size);

extern void *ExtModeCalloc(uint32_T number, uint32_T size);

#endif /* __MEM_MGR__ */

/* [EOF] mem_mgr.h */
```
